gfCNCPoint3[2431] = {X 27.2875, Y 32.6686, Z -3.8333, A 0.000, B 0.000, C 0.000 }
gfCNCPoint3[2432] = {X 27.6591, Y 33.1493, Z -3.8333, A 0.000, B 0.000, C 0.000 }
gfCNCPoint3[2433] = {X 27.9609, Y 33.6765, Z -3.8333, A 0.000, B 0.000, C 0.000 }
gfCNCPoint3[2434] = {X 30.9820, Y 39.9182, Z -3.8333, A 0.000, B 0.000, C 0.000 }
gfCNCPoint3[2435] = {X 31.3085, Y 40.8441, Z -3.8333, A 0.000, B 0.000, C 0.000 }
gfCNCPoint3[2436] = {X 31.4215, Y 41.8194, Z -3.8333, A 0.000, B 0.000, C 0.000 }
gfCNCPoint3[2437] = {X 31.3155, Y 42.7955, Z -3.8333, A 0.000, B 0.000, C 0.000 }
gfCNCPoint3[2438] = {X 30.9956, Y 43.7238, Z -3.8333, A 0.000, B 0.000, C 0.000 }
gfCNCPoint3[2439] = {X 30.4779, Y 44.5580, Z -3.8333, A 0.000, B 0.000, C 0.000 }
gfCNCPoint3[2440] = {X 29.7880, Y 45.2567, Z -3.8333, A 0.000, B 0.000, C 0.000 }
gfCNCPoint3[2441] = {X 29.2517, Y 45.6903, Z -3.8333, A 0.000, B 0.000, C 0.000 }
gfCNCPoint3[2442] = {X 28.5404, Y 46.1589, Z -3.8333, A 0.000, B 0.000, C 0.000 }
gfCNCPoint3[2443] = {X 27.7524, Y 46.4822, Z -3.8333, A 0.000, B 0.000, C 0.000 }
gfCNCPoint3[2444] = {X 26.9169, Y 46.6482, Z -3.8333, A 0.000, B 0.000, C 0.000 }
gfCNCPoint3[2445] = {X 26.0652, Y 46.6506, Z -3.8333, A 0.000, B 0.000, C 0.000 }
gfCNCPoint3[2446] = {X 25.2288, Y 46.4895, Z -3.8333, A 0.000, B 0.000, C 0.000 }
gfCNCPoint3[2447] = {X 23.4341, Y 47.4359, Z -3.8333, A 0.000, B 0.000, C 0.000 }
gfCNCPoint3[2448] = {X 21.5778, Y 48.2550, Z -3.8333, A 0.000, B 0.000, C 0.000 }
gfCNCPoint3[2449] = {X 19.6689, Y 48.9428, Z -3.8333, A 0.000, B 0.000, C 0.000 }
gfCNCPoint3[2450] = {X 19.5102, Y 48.9962, Z -3.8333, A 0.000, B 0.000, C 0.000 }
gfCNCPoint3[2451] = {X 17.3375, Y 49.5790, Z -3.8333, A 0.000, B 0.000, C 0.000 }
gfCNCPoint3[2452] = {X 15.1180, Y 49.9462, Z -3.8333, A 0.000, B 0.000, C 0.000 }
gfCNCPoint3[2453] = {X 12.8733, Y 50.0942, Z -3.8333, A 0.000, B 0.000, C 0.000 }
gfCNCPoint3[2454] = {X 10.6249, Y 50.0215, Z -3.8333, A 0.000, B 0.000, C 0.000 }
gfCNCPoint3[2455] = {X 8.3945, Y 49.7289, Z -3.8333, A 0.000, B 0.000, C 0.000 }
gfCNCPoint3[2456] = {X 6.6781, Y 49.3407, Z -3.8333, A 0.000, B 0.000, C 0.000 }
gfCNCPoint3[2457] = {X 5.0104, Y 48.7788, Z -3.8333, A 0.000, B 0.000, C 0.000 }
gfCNCPoint3[2458] = {X 3.4090, Y 48.0493, Z -3.8333, A 0.000, B 0.000, C 0.000 }
gfCNCPoint3[2459] = {X 2.3280, Y 47.4375, Z -3.8333, A 0.000, B 0.000, C 0.000 }
gfCNCPoint3[2460] = {X 1.2941, Y 46.7491, Z -3.8333, A 0.000, B 0.000, C 0.000 }
gfCNCPoint3[2461] = {X 0.5975, Y 46.2081, Z -3.8333, A 0.000, B 0.000, C 0.000 }
gfCNCPoint3[2462] = {X -0.5424, Y 45.1839, Z -3.8333, A 0.000, B 0.000, C 0.000 }
gfCNCPoint3[2463] = {X -1.5547, Y 44.0333, Z -3.8333, A 0.000, B 0.000, C 0.000 }
gfCNCPoint3[2464] = {X -2.4254, Y 42.7723, Z -3.8333, A 0.000, B 0.000, C 0.000 }
gfCNCPoint3[2465] = {X -3.1426, Y 41.4180, Z -3.8333, A 0.000, B 0.000, C 0.000 }
gfCNCPoint3[2466] = {X -3.6965, Y 39.9892, Z -3.8333, A 0.000, B 0.000, C 0.000 }
gfCNCPoint3[2467] = {X -3.6965, Y 41.3532, Z -3.8333, A 0.000, B 0.000, C 0.000 }
gfCNCPoint3[2468] = {X -3.0110, Y 42.7243, Z -3.8333, A 0.000, B 0.000, C 0.000 }
gfCNCPoint3[2469] = {X -2.1750, Y 44.0092, Z -3.8333, A 0.000, B 0.000, C 0.000 }
gfCNCPoint3[2470] = {X -1.1994, Y 45.1915, Z -3.8333, A 0.000, B 0.000, C 0.000 }
gfCNCPoint3[2471] = {X -0.0965, Y 46.2561, Z -3.8333, A 0.000, B 0.000, C 0.000 }
gfCNCPoint3[2472] = {X -0.0965, Y 99.1431, Z -3.8333, A 0.000, B 0.000, C 0.000 }
gfCNCPoint3[2473] = {X -0.0948, Y 100.0187, Z -3.8333, A 0.000, B 0.000, C 0.000 }
gfCNCPoint3[2474] = {X -0.0672, Y 100.0698, Z -3.8333, A 0.000, B 0.000, C 0.000 }
gfCNCPoint3[2475] = {X -0.0148, Y 100.0950, Z -3.8333, A 0.000, B 0.000, C 0.000 }
gfCNCPoint3[2476] = {X 120.5926, Y 100.0950, Z -3.8333, A 0.000, B 0.000, C 0.000 }
gfCNCPoint3[2477] = {X 121.0613, Y 100.8812, Z -3.8333, A 0.000, B 0.000, C 0.000 }
gfCNCPoint3[2478] = {X 121.6687, Y 101.5660, Z -3.8333, A 0.000, B 0.000, C 0.000 }
gfCNCPoint3[2479] = {X 122.3932, Y 102.1254, Z -3.8333, A 0.000, B 0.000, C 0.000 }
gfCNCPoint3[2480] = {X 123.2094, Y 102.5396, Z -3.8333, A 0.000, B 0.000, C 0.000 }
gfCNCPoint3[2481] = {X 124.0887, Y 102.7942, Z -3.8333, A 0.000, B 0.000, C 0.000 }
gfCNCPoint3[2482] = {X 125.0000, Y 102.8800, Z -3.8333, A 0.000, B 0.000, C 0.000 }
gfCNCPoint3[2483] = {X 143.7791, Y 102.8800, Z -3.8333, A 0.000, B 0.000, C 0.000 }
gfCNCPoint3[2484] = {X 144.6904, Y 102.7942, Z -3.8333, A 0.000, B 0.000, C 0.000 }
gfCNCPoint3[2485] = {X 145.5697, Y 102.5396, Z -3.8333, A 0.000, B 0.000, C 0.000 }
gfCNCPoint3[2486] = {X 146.3859, Y 102.1254, Z -3.8333, A 0.000, B 0.000, C 0.000 }
gfCNCPoint3[2487] = {X 147.1104, Y 101.5660, Z -3.8333, A 0.000, B 0.000, C 0.000 }
gfCNCPoint3[2488] = {X 147.7178, Y 100.8812, Z -3.8333, A 0.000, B 0.000, C 0.000 }
gfCNCPoint3[2489] = {X 148.1865, Y 100.0950, Z -3.8333, A 0.000, B 0.000, C 0.000 }
gfCNCPoint3[2490] = {X 150.8375, Y 100.0950, Z -3.8333, A 0.000, B 0.000, C 0.000 }
gfCNCPoint3[2491] = {X 150.8375, Y 95.2950, Z -3.8333, A 0.000, B 0.000, C 0.000 }
gfCNCPoint3[2492] = {X 187.9256, Y 95.2950, Z -3.8333, A 0.000, B 0.000, C 0.000 }
gfCNCPoint3[2493] = {X 187.9777, Y 95.0990, Z -3.8333, A 0.000, B 0.000, C 0.000 }
gfCNCPoint3[2494] = {X 188.0352, Y 94.9045, Z -3.8333, A 0.000, B 0.000, C 0.000 }
gfCNCPoint3[2495] = {X 187.2619, Y 94.0602, Z -3.8333, A 0.000, B 0.000, C 0.000 }
gfCNCPoint3[2496] = {X 151.4055, Y 94.0602, Z -3.8333, A 0.000, B 0.000, C 0.000 }
gfCNCPoint3[2497] = {X 150.7056, Y 94.8356, Z -3.8333, A 0.000, B 0.000, C 0.000 }
gfCNCPoint3[2498] = {X 150.7753, Y 95.0642, Z -3.8333, A 0.000, B 0.000, C 0.000 }
gfCNCPoint3[2499] = {X 150.8375, Y 95.2950, Z -3.8333, A 0.000, B 0.000, C 0.000 }
gfCNCPoint3[2500] = {X 150.8375, Y 97.6950, Z -3.8333, A 0.000, B 0.000, C 0.000 }
gfCNCPoint3[2501] = {X 190.1070, Y 97.6950, Z -3.8333, A 0.000, B 0.000, C 0.000 }
gfCNCPoint3[2502] = {X 190.1070, Y 97.0659, Z -3.8333, A 0.000, B 0.000, C 0.000 }
gfCNCPoint3[2503] = {X 190.1938, Y 96.1495, Z -3.8333, A 0.000, B 0.000, C 0.000 }
gfCNCPoint3[2504] = {X 190.4511, Y 95.2657, Z -3.8333, A 0.000, B 0.000, C 0.000 }
gfCNCPoint3[2505] = {X 190.8699, Y 94.4460, Z -3.8333, A 0.000, B 0.000, C 0.000 }
gfCNCPoint3[2506] = {X 188.3182, Y 91.6602, Z -3.8333, A 0.000, B 0.000, C 0.000 }
gfCNCPoint3[2507] = {X 150.3387, Y 91.6602, Z -3.8333, A 0.000, B 0.000, C 0.000 }
gfCNCPoint3[2508] = {X 147.8637, Y 94.4023, Z -3.8333, A 0.000, B 0.000, C 0.000 }
gfCNCPoint3[2509] = {X 148.2978, Y 95.2327, Z -3.8333, A 0.000, B 0.000, C 0.000 }
gfCNCPoint3[2510] = {X 148.5662, Y 96.1304, Z -3.8333, A 0.000, B 0.000, C 0.000 }
gfCNCPoint3[2511] = {X 148.6591, Y 97.0628, Z -3.8333, A 0.000, B 0.000, C 0.000 }
gfCNCPoint3[2512] = {X 148.6591, Y 97.6950, Z -3.8333, A 0.000, B 0.000, C 0.000 }
gfCNCPoint3[2513] = {X 150.8375, Y 97.6950, Z -3.8333, A 0.000, B 0.000, C 0.000 }
gfCNCPoint3[2514] = {X 150.8375, Y 100.0950, Z -3.8333, A 0.000, B 0.000, C 0.000 }
gfCNCPoint3[2515] = {X 190.5795, Y 100.0950, Z -3.8333, A 0.000, B 0.000, C 0.000 }
gfCNCPoint3[2516] = {X 191.0483, Y 100.8812, Z -3.8333, A 0.000, B 0.000, C 0.000 }
gfCNCPoint3[2517] = {X 191.6556, Y 101.5660, Z -3.8333, A 0.000, B 0.000, C 0.000 }
gfCNCPoint3[2518] = {X 192.3802, Y 102.1254, Z -3.8333, A 0.000, B 0.000, C 0.000 }
gfCNCPoint3[2519] = {X 193.1964, Y 102.5396, Z -3.8333, A 0.000, B 0.000, C 0.000 }
gfCNCPoint3[2520] = {X 194.0757, Y 102.7942, Z -3.8333, A 0.000, B 0.000, C 0.000 }
gfCNCPoint3[2521] = {X 194.9870, Y 102.8800, Z -3.8333, A 0.000, B 0.000, C 0.000 }
gfCNCPoint3[2522] = {X 212.6141, Y 102.8800, Z -3.8333, A 0.000, B 0.000, C 0.000 }
gfCNCPoint3[2523] = {X 213.0066, Y 102.8642, Z -3.8333, A 0.000, B 0.000, C 0.000 }
gfCNCPoint3[2524] = {X 213.3966, Y 102.8169, Z -3.8333, A 0.000, B 0.000, C 0.000 }
gfCNCPoint3[2525] = {X 213.7865, Y 102.8642, Z -3.8333, A 0.000, B 0.000, C 0.000 }
gfCNCPoint3[2526] = {X 214.1790, Y 102.8800, Z -3.8333, A 0.000, B 0.000, C 0.000 }
gfCNCPoint3[2527] = {X 233.4798, Y 102.8800, Z -3.8333, A 0.000, B 0.000, C 0.000 }
gfCNCPoint3[2528] = {X 234.3911, Y 102.7942, Z -3.8333, A 0.000, B 0.000, C 0.000 }
gfCNCPoint3[2529] = {X 235.2703, Y 102.5396, Z -3.8333, A 0.000, B 0.000, C 0.000 }
gfCNCPoint3[2530] = {X 236.0866, Y 102.1254, Z -3.8333, A 0.000, B 0.000, C 0.000 }
gfCNCPoint3[2531] = {X 236.8111, Y 101.5660, Z -3.8333, A 0.000, B 0.000, C 0.000 }
gfCNCPoint3[2532] = {X 237.4185, Y 100.8812, Z -3.8333, A 0.000, B 0.000, C 0.000 }
gfCNCPoint3[2533] = {X 237.8872, Y 100.0950, Z -3.8333, A 0.000, B 0.000, C 0.000 }
gfCNCPoint3[2534] = {X 261.4774, Y 100.0950, Z -3.8333, A 0.000, B 0.000, C 0.000 }
gfCNCPoint3[2535] = {X 261.4774, Y 90.4950, Z -3.8333, A 0.000, B 0.000, C 0.000 }
gfCNCPoint3[2536] = {X 266.0962, Y 90.4950, Z -3.8333, A 0.000, B 0.000, C 0.000 }
gfCNCPoint3[2537] = {X 266.1752, Y 90.3747, Z -3.8333, A 0.000, B 0.000, C 0.000 }
gfCNCPoint3[2538] = {X 266.2556, Y 90.2554, Z -3.8333, A 0.000, B 0.000, C 0.000 }
gfCNCPoint3[2539] = {X 263.5094, Y 89.1788, Z -3.8333, A 0.000, B 0.000, C 0.000 }
gfCNCPoint3[2540] = {X 261.4774, Y 90.4950, Z -3.8333, A 0.000, B 0.000, C 0.000 }
gfCNCPoint3[2541] = {X 261.4774, Y 92.8950, Z -3.8333, A 0.000, B 0.000, C 0.000 }
gfCNCPoint3[2542] = {X 267.4974, Y 92.8950, Z -3.8333, A 0.000, B 0.000, C 0.000 }
gfCNCPoint3[2543] = {X 267.8429, Y 92.2375, Z -3.8333, A 0.000, B 0.000, C 0.000 }
gfCNCPoint3[2544] = {X 268.2378, Y 91.6085, Z -3.8333, A 0.000, B 0.000, C 0.000 }
gfCNCPoint3[2545] = {X 269.1700, Y 90.4463, Z -3.8333, A 0.000, B 0.000, C 0.000 }
gfCNCPoint3[2546] = {X 270.2694, Y 89.4409, Z -3.8333, A 0.000, B 0.000, C 0.000 }
gfCNCPoint3[2547] = {X 270.2694, Y 89.2510, Z -3.8333, A 0.000, B 0.000, C 0.000 }
gfCNCPoint3[2548] = {X 263.2385, Y 86.4948, Z -3.8333, A 0.000, B 0.000, C 0.000 }
gfCNCPoint3[2549] = {X 253.3574, Y 92.8950, Z -3.8333, A 0.000, B 0.000, C 0.000 }
gfCNCPoint3[2550] = {X 261.4774, Y 92.8950, Z -3.8333, A 0.000, B 0.000, C 0.000 }
gfCNCPoint3[2551] = {X 261.4774, Y 95.2950, Z -3.8333, A 0.000, B 0.000, C 0.000 }
gfCNCPoint3[2552] = {X 269.1714, Y 95.2950, Z -3.8333, A 0.000, B 0.000, C 0.000 }
gfCNCPoint3[2553] = {X 269.5516, Y 94.1744, Z -3.8333, A 0.000, B 0.000, C 0.000 }
gfCNCPoint3[2554] = {X 270.1082, Y 93.1303, Z -3.8333, A 0.000, B 0.000, C 0.000 }
gfCNCPoint3[2555] = {X 270.8267, Y 92.1901, Z -3.8333, A 0.000, B 0.000, C 0.000 }
gfCNCPoint3[2556] = {X 271.6880, Y 91.3787, Z -3.8333, A 0.000, B 0.000, C 0.000 }
gfCNCPoint3[2557] = {X 272.6694, Y 90.7176, Z -3.8333, A 0.000, B 0.000, C 0.000 }
gfCNCPoint3[2558] = {X 272.6694, Y 87.6139, Z -3.8333, A 0.000, B 0.000, C 0.000 }
gfCNCPoint3[2559] = {X 262.9676, Y 83.8108, Z -3.8333, A 0.000, B 0.000, C 0.000 }
gfCNCPoint3[2560] = {X 245.2375, Y 95.2950, Z -3.8333, A 0.000, B 0.000, C 0.000 }
gfCNCPoint3[2561] = {X 261.4774, Y 95.2950, Z -3.8333, A 0.000, B 0.000, C 0.000 }
gfCNCPoint3[2562] = {X 261.4774, Y 97.6950, Z -3.8333, A 0.000, B 0.000, C 0.000 }
gfCNCPoint3[2563] = {X 271.3527, Y 97.6950, Z -3.8333, A 0.000, B 0.000, C 0.000 }
gfCNCPoint3[2564] = {X 271.3529, Y 97.0186, Z -3.8333, A 0.000, B 0.000, C 0.000 }
gfCNCPoint3[2565] = {X 271.4810, Y 95.9545, Z -3.8333, A 0.000, B 0.000, C 0.000 }
gfCNCPoint3[2566] = {X 271.8382, Y 94.9440, Z -3.8333, A 0.000, B 0.000, C 0.000 }
gfCNCPoint3[2567] = {X 272.4073, Y 94.0359, Z -3.8333, A 0.000, B 0.000, C 0.000 }
gfCNCPoint3[2568] = {X 273.1610, Y 93.2739, Z -3.8333, A 0.000, B 0.000, C 0.000 }
gfCNCPoint3[2569] = {X 274.0629, Y 92.6949, Z -3.8333, A 0.000, B 0.000, C 0.000 }
gfCNCPoint3[2570] = {X 275.0694, Y 92.3266, Z -3.8333, A 0.000, B 0.000, C 0.000 }
gfCNCPoint3[2571] = {X 275.0694, Y 85.9769, Z -3.8333, A 0.000, B 0.000, C 0.000 }
gfCNCPoint3[2572] = {X 262.6987, Y 81.1276, Z -3.8333, A 0.000, B 0.000, C 0.000 }
gfCNCPoint3[2573] = {X 262.5781, Y 81.2036, Z -3.8333, A 0.000, B 0.000, C 0.000 }
gfCNCPoint3[2574] = {X 238.3586, Y 96.8912, Z -3.8333, A 0.000, B 0.000, C 0.000 }
gfCNCPoint3[2575] = {X 238.3598, Y 97.0659, Z -3.8333, A 0.000, B 0.000, C 0.000 }
gfCNCPoint3[2576] = {X 238.3598, Y 97.6950, Z -3.8333, A 0.000, B 0.000, C 0.000 }
gfCNCPoint3[2577] = {X 261.4774, Y 97.6950, Z -3.8333, A 0.000, B 0.000, C 0.000 }
gfCNCPoint3[2578] = {X 261.4774, Y 100.0950, Z -3.8333, A 0.000, B 0.000, C 0.000 }
gfCNCPoint3[2579] = {X 271.8253, Y 100.0950, Z -3.8333, A 0.000, B 0.000, C 0.000 }
gfCNCPoint3[2580] = {X 272.2940, Y 100.8812, Z -3.8333, A 0.000, B 0.000, C 0.000 }
gfCNCPoint3[2581] = {X 272.9014, Y 101.5660, Z -3.8333, A 0.000, B 0.000, C 0.000 }
gfCNCPoint3[2582] = {X 273.6259, Y 102.1254, Z -3.8333, A 0.000, B 0.000, C 0.000 }
gfCNCPoint3[2583] = {X 274.4421, Y 102.5396, Z -3.8333, A 0.000, B 0.000, C 0.000 }
gfCNCPoint3[2584] = {X 275.3214, Y 102.7942, Z -3.8333, A 0.000, B 0.000, C 0.000 }
gfCNCPoint3[2585] = {X 276.2327, Y 102.8800, Z -3.8333, A 0.000, B 0.000, C 0.000 }
gfCNCPoint3[2586] = {X 292.7731, Y 102.8800, Z -3.8333, A 0.000, B 0.000, C 0.000 }
gfCNCPoint3[2587] = {X 293.6844, Y 102.7942, Z -3.8333, A 0.000, B 0.000, C 0.000 }
gfCNCPoint3[2588] = {X 294.5636, Y 102.5396, Z -3.8333, A 0.000, B 0.000, C 0.000 }
gfCNCPoint3[2589] = {X 295.3799, Y 102.1254, Z -3.8333, A 0.000, B 0.000, C 0.000 }
gfCNCPoint3[2590] = {X 296.1044, Y 101.5660, Z -3.8333, A 0.000, B 0.000, C 0.000 }
gfCNCPoint3[2591] = {X 296.7118, Y 100.8812, Z -3.8333, A 0.000, B 0.000, C 0.000 }
gfCNCPoint3[2592] = {X 297.1805, Y 100.0950, Z -3.8333, A 0.000, B 0.000, C 0.000 }
gfCNCPoint3[2593] = {X 319.1331, Y 100.0950, Z -3.8333, A 0.000, B 0.000, C 0.000 }
gfCNCPoint3[2594] = {X 321.4361, Y 100.8684, Z -3.8333, A 0.000, B 0.000, C 0.000 }
gfCNCPoint3[2595] = {X 323.7818, Y 101.5002, Z -3.8333, A 0.000, B 0.000, C 0.000 }
gfCNCPoint3[2596] = {X 326.1617, Y 101.9882, Z -3.8333, A 0.000, B 0.000, C 0.000 }
gfCNCPoint3[2597] = {X 329.6399, Y 102.5404, Z -3.8333, A 0.000, B 0.000, C 0.000 }
gfCNCPoint3[2598] = {X 333.1372, Y 102.9558, Z -3.8333, A 0.000, B 0.000, C 0.000 }
gfCNCPoint3[2599] = {X 336.6480, Y 103.2337, Z -3.8333, A 0.000, B 0.000, C 0.000 }
gfCNCPoint3[2600] = {X 342.8090, Y 103.5157, Z -3.8333, A 0.000, B 0.000, C 0.000 }
gfCNCPoint3[2601] = {X 348.9760, Y 103.5923, Z -3.8333, A 0.000, B 0.000, C 0.000 }
gfCNCPoint3[2602] = {X 355.1421, Y 103.4635, Z -3.8333, A 0.000, B 0.000, C 0.000 }
gfCNCPoint3[2603] = {X 361.3005, Y 103.1293, Z -3.8333, A 0.000, B 0.000, C 0.000 }
gfCNCPoint3[2604] = {X 365.1928, Y 102.7587, Z -3.8333, A 0.000, B 0.000, C 0.000 }
gfCNCPoint3[2605] = {X 369.0628, Y 102.2014, Z -3.8333, A 0.000, B 0.000, C 0.000 }
gfCNCPoint3[2606] = {X 372.9015, Y 101.4586, Z -3.8333, A 0.000, B 0.000, C 0.000 }
gfCNCPoint3[2607] = {X 375.2301, Y 100.8565, Z -3.8333, A 0.000, B 0.000, C 0.000 }
gfCNCPoint3[2608] = {X 377.5115, Y 100.0950, Z -3.8333, A 0.000, B 0.000, C 0.000 }
gfCNCPoint3[2609] = {X 391.9985, Y 100.0950, Z -3.8333, A 0.000, B 0.000, C 0.000 }
gfCNCPoint3[2610] = {X 392.4673, Y 100.8812, Z -3.8333, A 0.000, B 0.000, C 0.000 }
gfCNCPoint3[2611] = {X 393.0746, Y 101.5660, Z -3.8333, A 0.000, B 0.000, C 0.000 }
gfCNCPoint3[2612] = {X 393.7991, Y 102.1254, Z -3.8333, A 0.000, B 0.000, C 0.000 }
gfCNCPoint3[2613] = {X 394.6154, Y 102.5396, Z -3.8333, A 0.000, B 0.000, C 0.000 }
gfCNCPoint3[2614] = {X 395.4946, Y 102.7942, Z -3.8333, A 0.000, B 0.000, C 0.000 }
gfCNCPoint3[2615] = {X 396.4059, Y 102.8800, Z -3.8333, A 0.000, B 0.000, C 0.000 }
gfCNCPoint3[2616] = {X 415.7067, Y 102.8800, Z -3.8333, A 0.000, B 0.000, C 0.000 }
gfCNCPoint3[2617] = {X 416.6180, Y 102.7942, Z -3.8333, A 0.000, B 0.000, C 0.000 }
gfCNCPoint3[2618] = {X 417.4973, Y 102.5396, Z -3.8333, A 0.000, B 0.000, C 0.000 }
gfCNCPoint3[2619] = {X 418.3135, Y 102.1254, Z -3.8333, A 0.000, B 0.000, C 0.000 }
gfCNCPoint3[2620] = {X 419.0380, Y 101.5660, Z -3.8333, A 0.000, B 0.000, C 0.000 }
gfCNCPoint3[2621] = {X 419.6454, Y 100.8812, Z -3.8333, A 0.000, B 0.000, C 0.000 }
gfCNCPoint3[2622] = {X 420.1141, Y 100.0950, Z -3.8333, A 0.000, B 0.000, C 0.000 }
gfCNCPoint3[2623] = {X 443.7023, Y 100.0950, Z -3.8333, A 0.000, B 0.000, C 0.000 }
gfCNCPoint3[2624] = {X 443.7023, Y 90.4950, Z -3.8333, A 0.000, B 0.000, C 0.000 }
gfCNCPoint3[2625] = {X 448.3231, Y 90.4950, Z -3.8333, A 0.000, B 0.000, C 0.000 }
gfCNCPoint3[2626] = {X 448.4021, Y 90.3747, Z -3.8333, A 0.000, B 0.000, C 0.000 }
gfCNCPoint3[2627] = {X 448.4825, Y 90.2554, Z -3.8333, A 0.000, B 0.000, C 0.000 }
gfCNCPoint3[2628] = {X 445.7349, Y 89.1783, Z -3.8333, A 0.000, B 0.000, C 0.000 }
gfCNCPoint3[2629] = {X 443.7023, Y 90.4950, Z -3.8333, A 0.000, B 0.000, C 0.000 }
gfCNCPoint3[2630] = {X 443.7023, Y 92.8950, Z -3.8333, A 0.000, B 0.000, C 0.000 }
gfCNCPoint3[2631] = {X 449.7243, Y 92.8950, Z -3.8333, A 0.000, B 0.000, C 0.000 }
gfCNCPoint3[2632] = {X 450.0698, Y 92.2375, Z -3.8333, A 0.000, B 0.000, C 0.000 }
gfCNCPoint3[2633] = {X 450.4647, Y 91.6084, Z -3.8333, A 0.000, B 0.000, C 0.000 }
gfCNCPoint3[2634] = {X 451.3969, Y 90.4463, Z -3.8333, A 0.000, B 0.000, C 0.000 }
gfCNCPoint3[2635] = {X 452.4963, Y 89.4409, Z -3.8333, A 0.000, B 0.000, C 0.000 }
gfCNCPoint3[2636] = {X 452.4963, Y 89.2510, Z -3.8333, A 0.000, B 0.000, C 0.000 }
gfCNCPoint3[2637] = {X 445.4640, Y 86.4943, Z -3.8333, A 0.000, B 0.000, C 0.000 }
gfCNCPoint3[2638] = {X 435.5831, Y 92.8950, Z -3.8333, A 0.000, B 0.000, C 0.000 }
gfCNCPoint3[2639] = {X 443.7023, Y 92.8950, Z -3.8333, A 0.000, B 0.000, C 0.000 }
gfCNCPoint3[2640] = {X 443.7023, Y 95.2950, Z -3.8333, A 0.000, B 0.000, C 0.000 }
gfCNCPoint3[2641] = {X 451.3983, Y 95.2950, Z -3.8333, A 0.000, B 0.000, C 0.000 }
gfCNCPoint3[2642] = {X 451.7785, Y 94.1744, Z -3.8333, A 0.000, B 0.000, C 0.000 }
gfCNCPoint3[2643] = {X 452.3351, Y 93.1303, Z -3.8333, A 0.000, B 0.000, C 0.000 }
gfCNCPoint3[2644] = {X 453.0536, Y 92.1901, Z -3.8333, A 0.000, B 0.000, C 0.000 }
gfCNCPoint3[2645] = {X 453.9149, Y 91.3787, Z -3.8333, A 0.000, B 0.000, C 0.000 }
gfCNCPoint3[2646] = {X 454.8963, Y 90.7176, Z -3.8333, A 0.000, B 0.000, C 0.000 }
gfCNCPoint3[2647] = {X 454.8963, Y 87.6139, Z -3.8333, A 0.000, B 0.000, C 0.000 }
gfCNCPoint3[2648] = {X 445.1930, Y 83.8102, Z -3.8333, A 0.000, B 0.000, C 0.000 }
gfCNCPoint3[2649] = {X 427.4639, Y 95.2950, Z -3.8333, A 0.000, B 0.000, C 0.000 }
gfCNCPoint3[2650] = {X 443.7023, Y 95.2950, Z -3.8333, A 0.000, B 0.000, C 0.000 }
gfCNCPoint3[2651] = {X 443.7023, Y 97.6950, Z -3.8333, A 0.000, B 0.000, C 0.000 }
gfCNCPoint3[2652] = {X 453.5796, Y 97.6950, Z -3.8333, A 0.000, B 0.000, C 0.000 }
gfCNCPoint3[2653] = {X 453.5796, Y 97.0659, Z -3.8333, A 0.000, B 0.000, C 0.000 }
gfCNCPoint3[2654] = {X 453.6990, Y 95.9930, Z -3.8333, A 0.000, B 0.000, C 0.000 }
gfCNCPoint3[2655] = {X 454.0514, Y 94.9725, Z -3.8333, A 0.000, B 0.000, C 0.000 }
gfCNCPoint3[2656] = {X 454.6196, Y 94.0545, Z -3.8333, A 0.000, B 0.000, C 0.000 }
gfCNCPoint3[2657] = {X 455.3757, Y 93.2839, Z -3.8333, A 0.000, B 0.000, C 0.000 }
gfCNCPoint3[2658] = {X 456.2827, Y 92.6984, Z -3.8333, A 0.000, B 0.000, C 0.000 }
gfCNCPoint3[2659] = {X 457.2963, Y 92.3266, Z -3.8333, A 0.000, B 0.000, C 0.000 }
gfCNCPoint3[2660] = {X 457.2963, Y 85.9769, Z -3.8333, A 0.000, B 0.000, C 0.000 }
gfCNCPoint3[2661] = {X 444.9220, Y 81.1262, Z -3.8333, A 0.000, B 0.000, C 0.000 }
gfCNCPoint3[2662] = {X 420.5854, Y 96.8912, Z -3.8333, A 0.000, B 0.000, C 0.000 }
gfCNCPoint3[2663] = {X 420.5867, Y 97.0659, Z -3.8333, A 0.000, B 0.000, C 0.000 }
gfCNCPoint3[2664] = {X 420.5867, Y 97.6950, Z -3.8333, A 0.000, B 0.000, C 0.000 }
gfCNCPoint3[2665] = {X 443.7023, Y 97.6950, Z -3.8333, A 0.000, B 0.000, C 0.000 }
gfCNCPoint3[2666] = {X 443.7023, Y 100.0950, Z -3.8333, A 0.000, B 0.000, C 0.000 }
gfCNCPoint3[2667] = {X 454.0522, Y 100.0950, Z -3.8333, A 0.000, B 0.000, C 0.000 }
gfCNCPoint3[2668] = {X 454.5209, Y 100.8812, Z -3.8333, A 0.000, B 0.000, C 0.000 }
gfCNCPoint3[2669] = {X 455.1283, Y 101.5660, Z -3.8333, A 0.000, B 0.000, C 0.000 }
gfCNCPoint3[2670] = {X 455.8528, Y 102.1254, Z -3.8333, A 0.000, B 0.000, C 0.000 }
gfCNCPoint3[2671] = {X 456.6691, Y 102.5396, Z -3.8333, A 0.000, B 0.000, C 0.000 }
gfCNCPoint3[2672] = {X 457.5483, Y 102.7942, Z -3.8333, A 0.000, B 0.000, C 0.000 }
gfCNCPoint3[2673] = {X 458.4596, Y 102.8800, Z -3.8333, A 0.000, B 0.000, C 0.000 }
gfCNCPoint3[2674] = {X 475.0000, Y 102.8800, Z -3.8333, A 0.000, B 0.000, C 0.000 }
gfCNCPoint3[2675] = {X 475.9113, Y 102.7942, Z -3.8333, A 0.000, B 0.000, C 0.000 }
gfCNCPoint3[2676] = {X 476.7906, Y 102.5396, Z -3.8333, A 0.000, B 0.000, C 0.000 }
gfCNCPoint3[2677] = {X 477.6068, Y 102.1254, Z -3.8333, A 0.000, B 0.000, C 0.000 }
gfCNCPoint3[2678] = {X 478.3313, Y 101.5660, Z -3.8333, A 0.000, B 0.000, C 0.000 }
gfCNCPoint3[2679] = {X 478.9387, Y 100.8812, Z -3.8333, A 0.000, B 0.000, C 0.000 }
gfCNCPoint3[2680] = {X 479.4074, Y 100.0950, Z -3.8333, A 0.000, B 0.000, C 0.000 }
gfCNCPoint3[2681] = {X 507.6816, Y 100.0950, Z -3.8333, A 0.000, B 0.000, C 0.000 }
gfCNCPoint3[2682] = {X 507.6816, Y 107.6950, Z -3.8333, A 0.000, B 0.000, C 0.000 }
gfCNCPoint3[2683] = {X 507.6816, Y 107.6950, Z -0.8333, A 0.000, B 0.000, C 0.000 }
gfCNCPoint3[2684] = {X 507.6816, Y 107.6950, Z 11.0000, A 0.000, B 0.000, C 0.000 }
gfCNCPoint3[2685] = {X 108.5561, Y 40.8996, Z 11.0000, A 0.000, B 0.000, C 0.000 }
gfCNCPoint3[2686] = {X 108.5561, Y 40.8996, Z 0.0000, A 0.000, B 0.000, C 0.000 }
gfCNCPoint3[2687] = {X 108.5561, Y 40.8996, Z -3.8333, A 0.000, B 0.000, C 0.000 }
gfCNCPoint3[2688] = {X 108.0660, Y 42.0973, Z -3.8333, A 0.000, B 0.000, C 0.000 }
gfCNCPoint3[2689] = {X 108.0932, Y 42.0499, Z -3.8333, A 0.000, B 0.000, C 0.000 }
gfCNCPoint3[2690] = {X 108.1209, Y 42.0029, Z -3.8333, A 0.000, B 0.000, C 0.000 }
gfCNCPoint3[2691] = {X 108.5462, Y 41.3863, Z -3.8333, A 0.000, B 0.000, C 0.000 }
gfCNCPoint3[2692] = {X 109.0463, Y 40.8285, Z -3.8333, A 0.000, B 0.000, C 0.000 }
gfCNCPoint3[2693] = {X 109.0462, Y 39.7020, Z -3.8333, A 0.000, B 0.000, C 0.000 }
gfCNCPoint3[2694] = {X 108.5561, Y 40.8996, Z -3.8333, A 0.000, B 0.000, C 0.000 }
gfCNCPoint3[2695] = {X 108.5561, Y 40.8996, Z -0.8333, A 0.000, B 0.000, C 0.000 }
gfCNCPoint3[2696] = {X 108.5561, Y 40.8996, Z 11.0000, A 0.000, B 0.000, C 0.000 }
gfCNCPoint3[2697] = {X 95.6836, Y 40.8744, Z 11.0000, A 0.000, B 0.000, C 0.000 }
gfCNCPoint3[2698] = {X 95.6836, Y 40.8744, Z 0.0000, A 0.000, B 0.000, C 0.000 }
gfCNCPoint3[2699] = {X 95.6836, Y 40.8744, Z -3.8333, A 0.000, B 0.000, C 0.000 }
gfCNCPoint3[2700] = {X 95.2107, Y 39.7180, Z -3.8333, A 0.000, B 0.000, C 0.000 }
gfCNCPoint3[2701] = {X 95.2108, Y 40.8688, Z -3.8333, A 0.000, B 0.000, C 0.000 }
gfCNCPoint3[2702] = {X 95.7325, Y 41.4100, Z -3.8333, A 0.000, B 0.000, C 0.000 }
gfCNCPoint3[2703] = {X 96.1564, Y 42.0308, Z -3.8333, A 0.000, B 0.000, C 0.000 }
gfCNCPoint3[2704] = {X 95.6836, Y 40.8744, Z -3.8333, A 0.000, B 0.000, C 0.000 }
gfCNCPoint3[2705] = {X 95.6836, Y 40.8744, Z -0.8333, A 0.000, B 0.000, C 0.000 }
gfCNCPoint3[2706] = {X 95.6836, Y 40.8744, Z 11.0000, A 0.000, B 0.000, C 0.000 }
gfCNCPoint3[2707] = {X -7.6965, Y 43.3001, Z 11.0000, A 0.000, B 0.000, C 0.000 }
gfCNCPoint3[2708] = {X -7.6965, Y 43.3001, Z -0.8333, A 0.000, B 0.000, C 0.000 }
gfCNCPoint3[2709] = {X -7.6965, Y 43.3001, Z -3.8333, A 0.000, B 0.000, C 0.000 }
gfCNCPoint3[2710] = {X -3.6965, Y 30.8026, Z -3.8333, A 0.000, B 0.000, C 0.000 }
gfCNCPoint3[2711] = {X -3.5205, Y 30.2854, Z -3.8333, A 0.000, B 0.000, C 0.000 }
gfCNCPoint3[2712] = {X -3.3256, Y 29.7750, Z -3.8333, A 0.000, B 0.000, C 0.000 }
gfCNCPoint3[2713] = {X -2.7025, Y 28.4549, Z -3.8333, A 0.000, B 0.000, C 0.000 }
gfCNCPoint3[2714] = {X -1.9088, Y 27.2299, Z -3.8333, A 0.000, B 0.000, C 0.000 }
gfCNCPoint3[2715] = {X -0.9586, Y 26.1219, Z -3.8333, A 0.000, B 0.000, C 0.000 }
gfCNCPoint3[2716] = {X 0.1311, Y 25.1507, Z -3.8333, A 0.000, B 0.000, C 0.000 }
gfCNCPoint3[2717] = {X 1.3407, Y 24.3338, Z -3.8333, A 0.000, B 0.000, C 0.000 }
gfCNCPoint3[2718] = {X 0.5801, Y 23.9235, Z -3.8333, A 0.000, B 0.000, C 0.000 }
gfCNCPoint3[2719] = {X -0.0857, Y 23.3725, Z -3.8333, A 0.000, B 0.000, C 0.000 }
gfCNCPoint3[2720] = {X -0.6309, Y 22.7020, Z -3.8333, A 0.000, B 0.000, C 0.000 }
gfCNCPoint3[2721] = {X -1.0345, Y 21.9378, Z -3.8333, A 0.000, B 0.000, C 0.000 }
gfCNCPoint3[2722] = {X -3.6458, Y 15.5423, Z -3.8333, A 0.000, B 0.000, C 0.000 }
gfCNCPoint3[2723] = {X -3.6717, Y 15.4774, Z -3.8333, A 0.000, B 0.000, C 0.000 }
gfCNCPoint3[2724] = {X -3.6965, Y 15.4121, Z -3.8333, A 0.000, B 0.000, C 0.000 }
gfCNCPoint3[2725] = {X -7.6965, Y 4.6502, Z -3.8333, A 0.000, B 0.000, C 0.000 }
gfCNCPoint3[2726] = {X -7.6965, Y 4.6502, Z -0.8333, A 0.000, B 0.000, C 0.000 }
gfCNCPoint3[2727] = {X -7.6965, Y 4.6502, Z 11.0000, A 0.000, B 0.000, C 0.000 }
gfCNCPoint3[2728] = {X -7.6965, Y 16.4125, Z 11.0000, A 0.000, B 0.000, C 0.000 }
gfCNCPoint3[2729] = {X -7.6965, Y 16.4125, Z -0.8333, A 0.000, B 0.000, C 0.000 }
gfCNCPoint3[2730] = {X -7.6965, Y 16.4125, Z -3.8333, A 0.000, B 0.000, C 0.000 }
gfCNCPoint3[2731] = {X -4.8868, Y 16.4125, Z -3.8333, A 0.000, B 0.000, C 0.000 }
gfCNCPoint3[2732] = {X -3.6965, Y 12.5937, Z -3.8333, A 0.000, B 0.000, C 0.000 }
gfCNCPoint3[2733] = {X -3.6605, Y 12.4834, Z -3.8333, A 0.000, B 0.000, C 0.000 }
gfCNCPoint3[2734] = {X -3.6216, Y 12.3740, Z -3.8333, A 0.000, B 0.000, C 0.000 }
gfCNCPoint3[2735] = {X -3.1666, Y 11.4828, Z -3.8333, A 0.000, B 0.000, C 0.000 }
gfCNCPoint3[2736] = {X -2.5188, Y 10.7200, Z -3.8333, A 0.000, B 0.000, C 0.000 }
gfCNCPoint3[2737] = {X -1.7129, Y 10.1268, Z -3.8333, A 0.000, B 0.000, C 0.000 }
gfCNCPoint3[2738] = {X -1.1157, Y 9.7861, Z -3.8333, A 0.000, B 0.000, C 0.000 }
gfCNCPoint3[2739] = {X -0.2296, Y 9.4046, Z -3.8333, A 0.000, B 0.000, C 0.000 }
gfCNCPoint3[2740] = {X 0.7191, Y 9.2293, Z -3.8333, A 0.000, B 0.000, C 0.000 }
gfCNCPoint3[2741] = {X 1.6830, Y 9.2689, Z -3.8333, A 0.000, B 0.000, C 0.000 }
gfCNCPoint3[2742] = {X 2.6141, Y 9.5214, Z -3.8333, A 0.000, B 0.000, C 0.000 }
gfCNCPoint3[2743] = {X 3.3937, Y 9.1539, Z -3.8333, A 0.000, B 0.000, C 0.000 }
gfCNCPoint3[2744] = {X 4.1978, Y 8.8435, Z -3.8333, A 0.000, B 0.000, C 0.000 }
gfCNCPoint3[2745] = {X 6.1085, Y 8.1749, Z -3.8333, A 0.000, B 0.000, C 0.000 }
gfCNCPoint3[2746] = {X 8.0697, Y 7.6735, Z -3.8333, A 0.000, B 0.000, C 0.000 }
gfCNCPoint3[2747] = {X 10.0669, Y 7.3431, Z -3.8333, A 0.000, B 0.000, C 0.000 }
gfCNCPoint3[2748] = {X 12.0851, Y 7.1861, Z -3.8333, A 0.000, B 0.000, C 0.000 }
gfCNCPoint3[2749] = {X 14.1093, Y 7.2037, Z -3.8333, A 0.000, B 0.000, C 0.000 }
gfCNCPoint3[2750] = {X 16.1245, Y 7.3958, Z -3.8333, A 0.000, B 0.000, C 0.000 }
gfCNCPoint3[2751] = {X 17.9477, Y 7.7294, Z -3.8333, A 0.000, B 0.000, C 0.000 }
gfCNCPoint3[2752] = {X 19.7252, Y 8.2544, Z -3.8333, A 0.000, B 0.000, C 0.000 }
gfCNCPoint3[2753] = {X 21.4370, Y 8.9650, Z -3.8333, A 0.000, B 0.000, C 0.000 }
gfCNCPoint3[2754] = {X 23.0638, Y 9.8531, Z -3.8333, A 0.000, B 0.000, C 0.000 }
gfCNCPoint3[2755] = {X 24.5873, Y 10.9087, Z -3.8333, A 0.000, B 0.000, C 0.000 }
gfCNCPoint3[2756] = {X 25.6726, Y 11.8575, Z -3.8333, A 0.000, B 0.000, C 0.000 }
gfCNCPoint3[2757] = {X 26.6461, Y 12.9206, Z -3.8333, A 0.000, B 0.000, C 0.000 }
gfCNCPoint3[2758] = {X 27.4958, Y 14.0851, Z -3.8333, A 0.000, B 0.000, C 0.000 }
gfCNCPoint3[2759] = {X 28.2113, Y 15.3364, Z -3.8333, A 0.000, B 0.000, C 0.000 }
gfCNCPoint3[2760] = {X 28.7839, Y 16.6594, Z -3.8333, A 0.000, B 0.000, C 0.000 }
gfCNCPoint3[2761] = {X 29.2584, Y 18.3158, Z -3.8333, A 0.000, B 0.000, C 0.000 }
gfCNCPoint3[2762] = {X 29.5400, Y 20.0156, Z -3.8333, A 0.000, B 0.000, C 0.000 }
gfCNCPoint3[2763] = {X 29.6250, Y 21.7366, Z -3.8333, A 0.000, B 0.000, C 0.000 }
gfCNCPoint3[2764] = {X 29.5123, Y 23.4559, Z -3.8333, A 0.000, B 0.000, C 0.000 }
gfCNCPoint3[2765] = {X 29.2033, Y 25.1510, Z -3.8333, A 0.000, B 0.000, C 0.000 }
gfCNCPoint3[2766] = {X 28.7611, Y 26.5972, Z -3.8333, A 0.000, B 0.000, C 0.000 }
gfCNCPoint3[2767] = {X 28.1360, Y 27.9742, Z -3.8333, A 0.000, B 0.000, C 0.000 }
gfCNCPoint3[2768] = {X 27.3382, Y 29.2590, Z -3.8333, A 0.000, B 0.000, C 0.000 }
gfCNCPoint3[2769] = {X 26.3813, Y 30.4300, Z -3.8333, A 0.000, B 0.000, C 0.000 }
gfCNCPoint3[2770] = {X 25.2812, Y 31.4677, Z -3.8333, A 0.000, B 0.000, C 0.000 }
gfCNCPoint3[2771] = {X 26.0852, Y 31.8098, Z -3.8333, A 0.000, B 0.000, C 0.000 }
gfCNCPoint3[2772] = {X 26.8039, Y 32.3067, Z -3.8333, A 0.000, B 0.000, C 0.000 }
gfCNCPoint3[2773] = {X 27.4080, Y 32.9381, Z -3.8333, A 0.000, B 0.000, C 0.000 }
gfCNCPoint3[2774] = {X 27.8726, Y 33.6781, Z -3.8333, A 0.000, B 0.000, C 0.000 }
gfCNCPoint3[2775] = {X 30.9100, Y 39.9530, Z -3.8333, A 0.000, B 0.000, C 0.000 }
gfCNCPoint3[2776] = {X 31.2306, Y 40.8622, Z -3.8333, A 0.000, B 0.000, C 0.000 }
gfCNCPoint3[2777] = {X 31.3415, Y 41.8197, Z -3.8333, A 0.000, B 0.000, C 0.000 }
gfCNCPoint3[2778] = {X 31.2374, Y 42.7781, Z -3.8333, A 0.000, B 0.000, C 0.000 }
gfCNCPoint3[2779] = {X 30.9234, Y 43.6895, Z -3.8333, A 0.000, B 0.000, C 0.000 }
gfCNCPoint3[2780] = {X 30.4150, Y 44.5085, Z -3.8333, A 0.000, B 0.000, C 0.000 }
gfCNCPoint3[2781] = {X 29.7377, Y 45.1945, Z -3.8333, A 0.000, B 0.000, C 0.000 }
gfCNCPoint3[2782] = {X 29.2015, Y 45.6280, Z -3.8333, A 0.000, B 0.000, C 0.000 }
gfCNCPoint3[2783] = {X 28.4971, Y 46.0913, Z -3.8333, A 0.000, B 0.000, C 0.000 }
gfCNCPoint3[2784] = {X 27.7163, Y 46.4095, Z -3.8333, A 0.000, B 0.000, C 0.000 }
gfCNCPoint3[2785] = {X 26.8887, Y 46.5705, Z -3.8333, A 0.000, B 0.000, C 0.000 }
gfCNCPoint3[2786] = {X 26.0455, Y 46.5683, Z -3.8333, A 0.000, B 0.000, C 0.000 }
gfCNCPoint3[2787] = {X 25.2188, Y 46.4030, Z -3.8333, A 0.000, B 0.000, C 0.000 }
gfCNCPoint3[2788] = {X 23.4195, Y 47.3541, Z -3.8333, A 0.000, B 0.000, C 0.000 }
gfCNCPoint3[2789] = {X 21.5579, Y 48.1768, Z -3.8333, A 0.000, B 0.000, C 0.000 }
gfCNCPoint3[2790] = {X 19.6433, Y 48.8670, Z -3.8333, A 0.000, B 0.000, C 0.000 }
gfCNCPoint3[2791] = {X 17.4503, Y 49.4711, Z -3.8333, A 0.000, B 0.000, C 0.000 }
gfCNCPoint3[2792] = {X 15.2081, Y 49.8541, Z -3.8333, A 0.000, B 0.000, C 0.000 }
gfCNCPoint3[2793] = {X 12.9390, Y 50.0123, Z -3.8333, A 0.000, B 0.000, C 0.000 }
gfCNCPoint3[2794] = {X 10.6653, Y 49.9442, Z -3.8333, A 0.000, B 0.000, C 0.000 }
gfCNCPoint3[2795] = {X 8.4097, Y 49.6503, Z -3.8333, A 0.000, B 0.000, C 0.000 }
gfCNCPoint3[2796] = {X 6.5298, Y 49.2150, Z -3.8333, A 0.000, B 0.000, C 0.000 }
gfCNCPoint3[2797] = {X 4.7109, Y 48.5705, Z -3.8333, A 0.000, B 0.000, C 0.000 }
gfCNCPoint3[2798] = {X 2.9762, Y 47.7251, Z -3.8333, A 0.000, B 0.000, C 0.000 }
gfCNCPoint3[2799] = {X 1.3479, Y 46.6896, Z -3.8333, A 0.000, B 0.000, C 0.000 }
gfCNCPoint3[2800] = {X 0.6486, Y 46.1466, Z -3.8333, A 0.000, B 0.000, C 0.000 }
gfCNCPoint3[2801] = {X -0.4847, Y 45.1285, Z -3.8333, A 0.000, B 0.000, C 0.000 }
gfCNCPoint3[2802] = {X -1.4910, Y 43.9848, Z -3.8333, A 0.000, B 0.000, C 0.000 }
gfCNCPoint3[2803] = {X -2.3567, Y 42.7313, Z -3.8333, A 0.000, B 0.000, C 0.000 }
gfCNCPoint3[2804] = {X -3.0697, Y 41.3851, Z -3.8333, A 0.000, B 0.000, C 0.000 }
gfCNCPoint3[2805] = {X -3.6204, Y 39.9647, Z -3.8333, A 0.000, B 0.000, C 0.000 }
gfCNCPoint3[2806] = {X -3.6591, Y 39.8423, Z -3.8333, A 0.000, B 0.000, C 0.000 }
gfCNCPoint3[2807] = {X -3.6965, Y 39.7196, Z -3.8333, A 0.000, B 0.000, C 0.000 }
gfCNCPoint3[2808] = {X -4.8459, Y 35.8883, Z -3.8333, A 0.000, B 0.000, C 0.000 }
gfCNCPoint3[2809] = {X -7.9939, Y 36.0001, Z -3.8333, A 0.000, B 0.000, C 0.000 }
gfCNCPoint3[2810] = {X -7.9939, Y 36.0001, Z -0.8333, A 0.000, B 0.000, C 0.000 }
gfCNCPoint3[2811] = {X -7.9939, Y 36.0001, Z 11.0000, A 0.000, B 0.000, C 0.000 }
gfCNCPoint3[2812] = {X 608.0000, Y 40.1199, Z 11.0000, A 0.000, B 0.000, C 0.000 }
gfCNCPoint3[2813] = {X 608.0000, Y 40.1199, Z -0.8333, A 0.000, B 0.000, C 0.000 }
gfCNCPoint3[2814] = {X 608.0000, Y 40.1199, Z -3.8333, A 0.000, B 0.000, C 0.000 }
gfCNCPoint3[2815] = {X 603.6965, Y 47.2356, Z -3.8333, A 0.000, B 0.000, C 0.000 }
gfCNCPoint3[2816] = {X 603.6633, Y 47.2896, Z -3.8333, A 0.000, B 0.000, C 0.000 }
gfCNCPoint3[2817] = {X 603.6293, Y 47.3431, Z -3.8333, A 0.000, B 0.000, C 0.000 }
gfCNCPoint3[2818] = {X 603.0930, Y 48.0159, Z -3.8333, A 0.000, B 0.000, C 0.000 }
gfCNCPoint3[2819] = {X 602.4339, Y 48.5691, Z -3.8333, A 0.000, B 0.000, C 0.000 }
gfCNCPoint3[2820] = {X 601.6783, Y 48.9807, Z -3.8333, A 0.000, B 0.000, C 0.000 }
gfCNCPoint3[2821] = {X 600.8561, Y 49.2343, Z -3.8333, A 0.000, B 0.000, C 0.000 }
gfCNCPoint3[2822] = {X 600.0000, Y 49.3200, Z -3.8333, A 0.000, B 0.000, C 0.000 }
gfCNCPoint3[2823] = {X 593.5565, Y 49.3200, Z -3.8333, A 0.000, B 0.000, C 0.000 }
gfCNCPoint3[2824] = {X 592.5952, Y 49.2117, Z -3.8333, A 0.000, B 0.000, C 0.000 }
gfCNCPoint3[2825] = {X 591.6822, Y 48.8922, Z -3.8333, A 0.000, B 0.000, C 0.000 }
gfCNCPoint3[2826] = {X 590.8631, Y 48.3775, Z -3.8333, A 0.000, B 0.000, C 0.000 }
gfCNCPoint3[2827] = {X 590.1790, Y 47.6935, Z -3.8333, A 0.000, B 0.000, C 0.000 }
gfCNCPoint3[2828] = {X 589.6643, Y 46.8744, Z -3.8333, A 0.000, B 0.000, C 0.000 }
gfCNCPoint3[2829] = {X 589.3448, Y 45.9613, Z -3.8333, A 0.000, B 0.000, C 0.000 }
gfCNCPoint3[2830] = {X 589.2365, Y 45.0000, Z -3.8333, A 0.000, B 0.000, C 0.000 }
gfCNCPoint3[2831] = {X 589.2365, Y 44.0645, Z -3.8333, A 0.000, B 0.000, C 0.000 }
gfCNCPoint3[2832] = {X 589.3410, Y 43.1363, Z -3.8333, A 0.000, B 0.000, C 0.000 }
gfCNCPoint3[2833] = {X 589.6407, Y 42.2516, Z -3.8333, A 0.000, B 0.000, C 0.000 }
gfCNCPoint3[2834] = {X 590.1219, Y 41.4511, Z -3.8333, A 0.000, B 0.000, C 0.000 }
gfCNCPoint3[2835] = {X 590.7625, Y 40.7713, Z -3.8333, A 0.000, B 0.000, C 0.000 }
gfCNCPoint3[2836] = {X 590.7630, Y 33.5305, Z -3.8333, A 0.000, B 0.000, C 0.000 }
gfCNCPoint3[2837] = {X 585.4453, Y 46.6524, Z -3.8333, A 0.000, B 0.000, C 0.000 }
gfCNCPoint3[2838] = {X 585.0755, Y 47.3550, Z -3.8333, A 0.000, B 0.000, C 0.000 }
gfCNCPoint3[2839] = {X 584.5834, Y 47.9780, Z -3.8333, A 0.000, B 0.000, C 0.000 }
gfCNCPoint3[2840] = {X 583.9856, Y 48.5004, Z -3.8333, A 0.000, B 0.000, C 0.000 }
gfCNCPoint3[2841] = {X 583.3023, Y 48.9046, Z -3.8333, A 0.000, B 0.000, C 0.000 }
gfCNCPoint3[2842] = {X 582.3585, Y 49.2242, Z -3.8333, A 0.000, B 0.000, C 0.000 }
gfCNCPoint3[2843] = {X 581.3666, Y 49.3191, Z -3.8333, A 0.000, B 0.000, C 0.000 }
gfCNCPoint3[2844] = {X 580.3794, Y 49.1842, Z -3.8333, A 0.000, B 0.000, C 0.000 }
gfCNCPoint3[2845] = {X 579.4493, Y 48.8268, Z -3.8333, A 0.000, B 0.000, C 0.000 }
gfCNCPoint3[2846] = {X 578.6259, Y 48.2657, Z -3.8333, A 0.000, B 0.000, C 0.000 }
gfCNCPoint3[2847] = {X 577.9529, Y 47.5309, Z -3.8333, A 0.000, B 0.000, C 0.000 }
gfCNCPoint3[2848] = {X 577.4662, Y 46.6615, Z -3.8333, A 0.000, B 0.000, C 0.000 }
gfCNCPoint3[2849] = {X 572.0186, Y 33.3407, Z -3.8333, A 0.000, B 0.000, C 0.000 }
gfCNCPoint3[2850] = {X 572.0189, Y 40.7699, Z -3.8333, A 0.000, B 0.000, C 0.000 }
gfCNCPoint3[2851] = {X 572.6574, Y 41.4410, Z -3.8333, A 0.000, B 0.000, C 0.000 }
gfCNCPoint3[2852] = {X 573.1381, Y 42.2327, Z -3.8333, A 0.000, B 0.000, C 0.000 }
gfCNCPoint3[2853] = {X 573.4390, Y 43.1087, Z -3.8333, A 0.000, B 0.000, C 0.000 }
gfCNCPoint3[2854] = {X 573.5463, Y 44.0287, Z -3.8333, A 0.000, B 0.000, C 0.000 }
gfCNCPoint3[2855] = {X 573.5464, Y 45.0000, Z -3.8333, A 0.000, B 0.000, C 0.000 }
gfCNCPoint3[2856] = {X 573.4381, Y 45.9613, Z -3.8333, A 0.000, B 0.000, C 0.000 }
gfCNCPoint3[2857] = {X 573.1186, Y 46.8744, Z -3.8333, A 0.000, B 0.000, C 0.000 }
gfCNCPoint3[2858] = {X 572.6039, Y 47.6935, Z -3.8333, A 0.000, B 0.000, C 0.000 }
gfCNCPoint3[2859] = {X 571.9199, Y 48.3775, Z -3.8333, A 0.000, B 0.000, C 0.000 }
gfCNCPoint3[2860] = {X 571.1008, Y 48.8922, Z -3.8333, A 0.000, B 0.000, C 0.000 }
gfCNCPoint3[2861] = {X 570.1877, Y 49.2117, Z -3.8333, A 0.000, B 0.000, C 0.000 }
gfCNCPoint3[2862] = {X 569.2264, Y 49.3200, Z -3.8333, A 0.000, B 0.000, C 0.000 }
gfCNCPoint3[2863] = {X 562.4443, Y 49.3200, Z -3.8333, A 0.000, B 0.000, C 0.000 }
gfCNCPoint3[2864] = {X 561.4830, Y 49.2117, Z -3.8333, A 0.000, B 0.000, C 0.000 }
gfCNCPoint3[2865] = {X 560.5699, Y 48.8922, Z -3.8333, A 0.000, B 0.000, C 0.000 }
gfCNCPoint3[2866] = {X 559.7508, Y 48.3775, Z -3.8333, A 0.000, B 0.000, C 0.000 }
gfCNCPoint3[2867] = {X 559.0668, Y 47.6935, Z -3.8333, A 0.000, B 0.000, C 0.000 }
gfCNCPoint3[2868] = {X 558.5521, Y 46.8744, Z -3.8333, A 0.000, B 0.000, C 0.000 }
gfCNCPoint3[2869] = {X 558.2326, Y 45.9613, Z -3.8333, A 0.000, B 0.000, C 0.000 }
gfCNCPoint3[2870] = {X 558.1243, Y 45.0000, Z -3.8333, A 0.000, B 0.000, C 0.000 }
gfCNCPoint3[2871] = {X 558.1243, Y 44.0646, Z -3.8333, A 0.000, B 0.000, C 0.000 }
gfCNCPoint3[2872] = {X 558.2286, Y 43.1360, Z -3.8333, A 0.000, B 0.000, C 0.000 }
gfCNCPoint3[2873] = {X 558.5286, Y 42.2510, Z -3.8333, A 0.000, B 0.000, C 0.000 }
gfCNCPoint3[2874] = {X 559.0105, Y 41.4504, Z -3.8333, A 0.000, B 0.000, C 0.000 }
gfCNCPoint3[2875] = {X 559.6521, Y 40.7710, Z -3.8333, A 0.000, B 0.000, C 0.000 }
gfCNCPoint3[2876] = {X 559.6521, Y 9.2304, Z -3.8333, A 0.000, B 0.000, C 0.000 }
gfCNCPoint3[2877] = {X 559.0136, Y 8.5594, Z -3.8333, A 0.000, B 0.000, C 0.000 }
gfCNCPoint3[2878] = {X 558.5328, Y 7.7678, Z -3.8333, A 0.000, B 0.000, C 0.000 }
gfCNCPoint3[2879] = {X 558.2318, Y 6.8918, Z -3.8333, A 0.000, B 0.000, C 0.000 }
gfCNCPoint3[2880] = {X 558.1245, Y 5.9718, Z -3.8333, A 0.000, B 0.000, C 0.000 }
gfCNCPoint3[2881] = {X 558.1243, Y 5.0000, Z -3.8333, A 0.000, B 0.000, C 0.000 }
gfCNCPoint3[2882] = {X 558.2326, Y 4.0387, Z -3.8333, A 0.000, B 0.000, C 0.000 }
gfCNCPoint3[2883] = {X 558.5521, Y 3.1256, Z -3.8333, A 0.000, B 0.000, C 0.000 }
gfCNCPoint3[2884] = {X 559.0668, Y 2.3065, Z -3.8333, A 0.000, B 0.000, C 0.000 }
gfCNCPoint3[2885] = {X 559.7508, Y 1.6225, Z -3.8333, A 0.000, B 0.000, C 0.000 }
gfCNCPoint3[2886] = {X 560.5699, Y 1.1078, Z -3.8333, A 0.000, B 0.000, C 0.000 }
gfCNCPoint3[2887] = {X 561.4830, Y 0.7883, Z -3.8333, A 0.000, B 0.000, C 0.000 }
gfCNCPoint3[2888] = {X 562.4443, Y 0.6800, Z -3.8333, A 0.000, B 0.000, C 0.000 }
gfCNCPoint3[2889] = {X 570.9376, Y 0.6800, Z -3.8333, A 0.000, B 0.000, C 0.000 }
gfCNCPoint3[2890] = {X 571.8988, Y 0.7883, Z -3.8333, A 0.000, B 0.000, C 0.000 }
gfCNCPoint3[2891] = {X 572.8119, Y 1.1078, Z -3.8333, A 0.000, B 0.000, C 0.000 }
gfCNCPoint3[2892] = {X 573.6310, Y 1.6225, Z -3.8333, A 0.000, B 0.000, C 0.000 }
gfCNCPoint3[2893] = {X 574.3151, Y 2.3065, Z -3.8333, A 0.000, B 0.000, C 0.000 }
gfCNCPoint3[2894] = {X 574.8297, Y 3.1256, Z -3.8333, A 0.000, B 0.000, C 0.000 }
gfCNCPoint3[2895] = {X 575.1492, Y 4.0387, Z -3.8333, A 0.000, B 0.000, C 0.000 }
gfCNCPoint3[2896] = {X 575.2576, Y 5.0000, Z -3.8333, A 0.000, B 0.000, C 0.000 }
gfCNCPoint3[2897] = {X 575.2576, Y 5.9342, Z -3.8333, A 0.000, B 0.000, C 0.000 }
gfCNCPoint3[2898] = {X 575.1835, Y 6.7306, Z -3.8333, A 0.000, B 0.000, C 0.000 }
gfCNCPoint3[2899] = {X 574.9638, Y 7.4998, Z -3.8333, A 0.000, B 0.000, C 0.000 }
gfCNCPoint3[2900] = {X 574.6062, Y 8.2152, Z -3.8333, A 0.000, B 0.000, C 0.000 }
gfCNCPoint3[2901] = {X 581.1909, Y 24.3702, Z -3.8333, A 0.000, B 0.000, C 0.000 }
gfCNCPoint3[2902] = {X 587.8458, Y 8.0943, Z -3.8333, A 0.000, B 0.000, C 0.000 }
gfCNCPoint3[2903] = {X 587.5317, Y 7.4231, Z -3.8333, A 0.000, B 0.000, C 0.000 }
gfCNCPoint3[2904] = {X 587.3369, Y 6.7082, Z -3.8333, A 0.000, B 0.000, C 0.000 }
gfCNCPoint3[2905] = {X 587.2671, Y 5.9705, Z -3.8333, A 0.000, B 0.000, C 0.000 }
gfCNCPoint3[2906] = {X 587.2670, Y 5.0000, Z -3.8333, A 0.000, B 0.000, C 0.000 }
gfCNCPoint3[2907] = {X 587.3753, Y 4.0387, Z -3.8333, A 0.000, B 0.000, C 0.000 }
gfCNCPoint3[2908] = {X 587.6948, Y 3.1256, Z -3.8333, A 0.000, B 0.000, C 0.000 }
gfCNCPoint3[2909] = {X 588.2094, Y 2.3065, Z -3.8333, A 0.000, B 0.000, C 0.000 }
gfCNCPoint3[2910] = {X 588.8935, Y 1.6225, Z -3.8333, A 0.000, B 0.000, C 0.000 }
gfCNCPoint3[2911] = {X 589.7126, Y 1.1078, Z -3.8333, A 0.000, B 0.000, C 0.000 }
gfCNCPoint3[2912] = {X 590.6257, Y 0.7883, Z -3.8333, A 0.000, B 0.000, C 0.000 }
gfCNCPoint3[2913] = {X 591.5870, Y 0.6800, Z -3.8333, A 0.000, B 0.000, C 0.000 }
gfCNCPoint3[2914] = {X 600.0000, Y 0.6800, Z -3.8333, A 0.000, B 0.000, C 0.000 }
gfCNCPoint3[2915] = {X 600.8561, Y 0.7657, Z -3.8333, A 0.000, B 0.000, C 0.000 }
gfCNCPoint3[2916] = {X 601.6783, Y 1.0193, Z -3.8333, A 0.000, B 0.000, C 0.000 }
gfCNCPoint3[2917] = {X 602.4339, Y 1.4309, Z -3.8333, A 0.000, B 0.000, C 0.000 }
gfCNCPoint3[2918] = {X 603.0930, Y 1.9841, Z -3.8333, A 0.000, B 0.000, C 0.000 }
gfCNCPoint3[2919] = {X 603.6293, Y 2.6569, Z -3.8333, A 0.000, B 0.000, C 0.000 }
gfCNCPoint3[2920] = {X 603.6633, Y 2.7104, Z -3.8333, A 0.000, B 0.000, C 0.000 }
gfCNCPoint3[2921] = {X 603.6965, Y 2.7644, Z -3.8333, A 0.000, B 0.000, C 0.000 }
gfCNCPoint3[2922] = {X 608.0000, Y 9.8801, Z -3.8333, A 0.000, B 0.000, C 0.000 }
gfCNCPoint3[2923] = {X 608.0000, Y 9.8801, Z -0.8333, A 0.000, B 0.000, C 0.000 }
gfCNCPoint3[2924] = {X 608.0000, Y 9.8801, Z 11.0000, A 0.000, B 0.000, C 0.000 }
gfCNCPoint3[2925] = {X -7.6965, Y 16.7864, Z 11.0000, A 0.000, B 0.000, C 0.000 }
gfCNCPoint3[2926] = {X -7.6965, Y 16.7864, Z -0.8333, A 0.000, B 0.000, C 0.000 }
gfCNCPoint3[2927] = {X -7.6965, Y 16.7864, Z -3.8333, A 0.000, B 0.000, C 0.000 }
gfCNCPoint3[2928] = {X -4.6245, Y 16.7864, Z -3.8333, A 0.000, B 0.000, C 0.000 }
gfCNCPoint3[2929] = {X -3.6965, Y 12.8955, Z -3.8333, A 0.000, B 0.000, C 0.000 }
gfCNCPoint3[2930] = {X -3.6291, Y 12.6464, Z -3.8333, A 0.000, B 0.000, C 0.000 }
gfCNCPoint3[2931] = {X -3.5466, Y 12.4019, Z -3.8333, A 0.000, B 0.000, C 0.000 }
gfCNCPoint3[2932] = {X -3.1001, Y 11.5271, Z -3.8333, A 0.000, B 0.000, C 0.000 }
gfCNCPoint3[2933] = {X -2.4643, Y 10.7785, Z -3.8333, A 0.000, B 0.000, C 0.000 }
gfCNCPoint3[2934] = {X -1.6733, Y 10.1963, Z -3.8333, A 0.000, B 0.000, C 0.000 }
gfCNCPoint3[2935] = {X -1.0760, Y 9.8556, Z -3.8333, A 0.000, B 0.000, C 0.000 }
gfCNCPoint3[2936] = {X -0.1977, Y 9.4785, Z -3.8333, A 0.000, B 0.000, C 0.000 }
gfCNCPoint3[2937] = {X 0.7428, Y 9.3079, Z -3.8333, A 0.000, B 0.000, C 0.000 }
gfCNCPoint3[2938] = {X 1.6977, Y 9.3522, Z -3.8333, A 0.000, B 0.000, C 0.000 }
gfCNCPoint3[2939] = {X 2.6183, Y 9.6093, Z -3.8333, A 0.000, B 0.000, C 0.000 }
gfCNCPoint3[2940] = {X 3.4093, Y 9.2342, Z -3.8333, A 0.000, B 0.000, C 0.000 }
gfCNCPoint3[2941] = {X 4.2257, Y 8.9185, Z -3.8333, A 0.000, B 0.000, C 0.000 }
gfCNCPoint3[2942] = {X 6.1302, Y 8.2519, Z -3.8333, A 0.000, B 0.000, C 0.000 }
gfCNCPoint3[2943] = {X 8.0851, Y 7.7520, Z -3.8333, A 0.000, B 0.000, C 0.000 }
gfCNCPoint3[2944] = {X 10.0758, Y 7.4226, Z -3.8333, A 0.000, B 0.000, C 0.000 }
gfCNCPoint3[2945] = {X 12.0875, Y 7.2661, Z -3.8333, A 0.000, B 0.000, C 0.000 }
gfCNCPoint3[2946] = {X 14.1052, Y 7.2836, Z -3.8333, A 0.000, B 0.000, C 0.000 }
gfCNCPoint3[2947] = {X 16.1139, Y 7.4751, Z -3.8333, A 0.000, B 0.000, C 0.000 }
gfCNCPoint3[2948] = {X 17.9288, Y 7.8071, Z -3.8333, A 0.000, B 0.000, C 0.000 }
gfCNCPoint3[2949] = {X 19.6982, Y 8.3298, Z -3.8333, A 0.000, B 0.000, C 0.000 }
gfCNCPoint3[2950] = {X 21.4023, Y 9.0371, Z -3.8333, A 0.000, B 0.000, C 0.000 }
gfCNCPoint3[2951] = {X 23.0218, Y 9.9211, Z -3.8333, A 0.000, B 0.000, C 0.000 }
gfCNCPoint3[2952] = {X 24.5383, Y 10.9719, Z -3.8333, A 0.000, B 0.000, C 0.000 }
gfCNCPoint3[2953] = {X 25.6168, Y 11.9148, Z -3.8333, A 0.000, B 0.000, C 0.000 }
gfCNCPoint3[2954] = {X 26.5843, Y 12.9714, Z -3.8333, A 0.000, B 0.000, C 0.000 }
gfCNCPoint3[2955] = {X 27.4287, Y 14.1287, Z -3.8333, A 0.000, B 0.000, C 0.000 }
gfCNCPoint3[2956] = {X 28.1398, Y 15.3723, Z -3.8333, A 0.000, B 0.000, C 0.000 }
gfCNCPoint3[2957] = {X 28.7088, Y 16.6870, Z -3.8333, A 0.000, B 0.000, C 0.000 }
gfCNCPoint3[2958] = {X 29.1806, Y 18.3344, Z -3.8333, A 0.000, B 0.000, C 0.000 }
gfCNCPoint3[2959] = {X 29.4606, Y 20.0250, Z -3.8333, A 0.000, B 0.000, C 0.000 }
gfCNCPoint3[2960] = {X 29.5450, Y 21.7366, Z -3.8333, A 0.000, B 0.000, C 0.000 }
gfCNCPoint3[2961] = {X 29.4329, Y 23.4465, Z -3.8333, A 0.000, B 0.000, C 0.000 }
gfCNCPoint3[2962] = {X 29.1255, Y 25.1324, Z -3.8333, A 0.000, B 0.000, C 0.000 }
gfCNCPoint3[2963] = {X 28.6756, Y 26.5971, Z -3.8333, A 0.000, B 0.000, C 0.000 }
gfCNCPoint3[2964] = {X 28.0367, Y 27.9898, Z -3.8333, A 0.000, B 0.000, C 0.000 }
gfCNCPoint3[2965] = {X 27.2200, Y 29.2862, Z -3.8333, A 0.000, B 0.000, C 0.000 }
gfCNCPoint3[2966] = {X 26.2397, Y 30.4637, Z -3.8333, A 0.000, B 0.000, C 0.000 }
gfCNCPoint3[2967] = {X 25.1128, Y 31.5019, Z -3.8333, A 0.000, B 0.000, C 0.000 }
gfCNCPoint3[2968] = {X 25.2523, Y 31.5425, Z -3.8333, A 0.000, B 0.000, C 0.000 }
gfCNCPoint3[2969] = {X 25.3904, Y 31.5877, Z -3.8333, A 0.000, B 0.000, C 0.000 }
gfCNCPoint3[2970] = {X 26.1379, Y 31.9316, Z -3.8333, A 0.000, B 0.000, C 0.000 }
gfCNCPoint3[2971] = {X 26.8049, Y 32.4134, Z -3.8333, A 0.000, B 0.000, C 0.000 }
gfCNCPoint3[2972] = {X 27.3662, Y 33.0150, Z -3.8333, A 0.000, B 0.000, C 0.000 }
gfCNCPoint3[2973] = {X 27.8009, Y 33.7136, Z -3.8333, A 0.000, B 0.000, C 0.000 }
gfCNCPoint3[2974] = {X 30.8380, Y 39.9879, Z -3.8333, A 0.000, B 0.000, C 0.000 }
gfCNCPoint3[2975] = {X 31.1526, Y 40.8802, Z -3.8333, A 0.000, B 0.000, C 0.000 }
gfCNCPoint3[2976] = {X 31.2615, Y 41.8200, Z -3.8333, A 0.000, B 0.000, C 0.000 }
gfCNCPoint3[2977] = {X 31.1593, Y 42.7606, Z -3.8333, A 0.000, B 0.000, C 0.000 }
gfCNCPoint3[2978] = {X 30.8511, Y 43.6551, Z -3.8333, A 0.000, B 0.000, C 0.000 }
gfCNCPoint3[2979] = {X 30.3522, Y 44.4590, Z -3.8333, A 0.000, B 0.000, C 0.000 }
gfCNCPoint3[2980] = {X 29.6874, Y 45.1323, Z -3.8333, A 0.000, B 0.000, C 0.000 }
gfCNCPoint3[2981] = {X 29.1512, Y 45.5658, Z -3.8333, A 0.000, B 0.000, C 0.000 }
gfCNCPoint3[2982] = {X 28.4537, Y 46.0237, Z -3.8333, A 0.000, B 0.000, C 0.000 }
gfCNCPoint3[2983] = {X 27.6802, Y 46.3368, Z -3.8333, A 0.000, B 0.000, C 0.000 }
gfCNCPoint3[2984] = {X 26.8605, Y 46.4928, Z -3.8333, A 0.000, B 0.000, C 0.000 }
gfCNCPoint3[2985] = {X 26.0261, Y 46.4859, Z -3.8333, A 0.000, B 0.000, C 0.000 }
gfCNCPoint3[2986] = {X 25.2091, Y 46.3163, Z -3.8333, A 0.000, B 0.000, C 0.000 }
gfCNCPoint3[2987] = {X 23.4053, Y 47.2720, Z -3.8333, A 0.000, B 0.000, C 0.000 }
gfCNCPoint3[2988] = {X 21.5387, Y 48.0983, Z -3.8333, A 0.000, B 0.000, C 0.000 }
gfCNCPoint3[2989] = {X 19.6186, Y 48.7909, Z -3.8333, A 0.000, B 0.000, C 0.000 }
gfCNCPoint3[2990] = {X 17.4331, Y 49.3929, Z -3.8333, A 0.000, B 0.000, C 0.000 }
gfCNCPoint3[2991] = {X 15.1987, Y 49.7747, Z -3.8333, A 0.000, B 0.000, C 0.000 }
gfCNCPoint3[2992] = {X 12.9373, Y 49.9324, Z -3.8333, A 0.000, B 0.000, C 0.000 }
gfCNCPoint3[2993] = {X 10.6715, Y 49.8644, Z -3.8333, A 0.000, B 0.000, C 0.000 }
gfCNCPoint3[2994] = {X 8.4237, Y 49.5716, Z -3.8333, A 0.000, B 0.000, C 0.000 }
gfCNCPoint3[2995] = {X 6.5528, Y 49.1384, Z -3.8333, A 0.000, B 0.000, C 0.000 }
gfCNCPoint3[2996] = {X 4.7427, Y 48.4971, Z -3.8333, A 0.000, B 0.000, C 0.000 }
gfCNCPoint3[2997] = {X 3.0163, Y 47.6559, Z -3.8333, A 0.000, B 0.000, C 0.000 }
gfCNCPoint3[2998] = {X 1.3958, Y 46.6255, Z -3.8333, A 0.000, B 0.000, C 0.000 }
gfCNCPoint3[2999] = {X 0.6985, Y 46.0840, Z -3.8333, A 0.000, B 0.000, C 0.000 }
gfCNCPoint3[3000] = {X -0.4278, Y 45.0722, Z -3.8333, A 0.000, B 0.000, C 0.000 }
gfCNCPoint3[3001] = {X -1.4280, Y 43.9356, Z -3.8333, A 0.000, B 0.000, C 0.000 }
gfCNCPoint3[3002] = {X -2.2883, Y 42.6898, Z -3.8333, A 0.000, B 0.000, C 0.000 }
gfCNCPoint3[3003] = {X -2.9970, Y 41.3518, Z -3.8333, A 0.000, B 0.000, C 0.000 }
gfCNCPoint3[3004] = {X -3.5442, Y 39.9402, Z -3.8333, A 0.000, B 0.000, C 0.000 }
gfCNCPoint3[3005] = {X -3.6230, Y 39.6863, Z -3.8333, A 0.000, B 0.000, C 0.000 }
gfCNCPoint3[3006] = {X -3.6965, Y 39.4309, Z -3.8333, A 0.000, B 0.000, C 0.000 }
gfCNCPoint3[3007] = {X -4.7636, Y 35.5759, Z -3.8333, A 0.000, B 0.000, C 0.000 }
gfCNCPoint3[3008] = {X -8.0034, Y 35.6252, Z -3.8333, A 0.000, B 0.000, C 0.000 }
gfCNCPoint3[3009] = {X -8.0034, Y 35.6252, Z -0.8333, A 0.000, B 0.000, C 0.000 }
gfCNCPoint3[3010] = {X -8.0034, Y 35.6252, Z 11.0000, A 0.000, B 0.000, C 0.000 }
gfCNCPoint3[3011] = {X -7.6965, Y 17.3012, Z 11.0000, A 0.000, B 0.000, C 0.000 }
gfCNCPoint3[3012] = {X -7.6965, Y 17.3012, Z -0.8333, A 0.000, B 0.000, C 0.000 }
gfCNCPoint3[3013] = {X -7.6965, Y 17.3012, Z -3.8333, A 0.000, B 0.000, C 0.000 }
gfCNCPoint3[3014] = {X -4.2193, Y 17.3012, Z -3.8333, A 0.000, B 0.000, C 0.000 }
gfCNCPoint3[3015] = {X -3.6965, Y 13.3355, Z -3.8333, A 0.000, B 0.000, C 0.000 }
gfCNCPoint3[3016] = {X -3.6095, Y 12.8763, Z -3.8333, A 0.000, B 0.000, C 0.000 }
gfCNCPoint3[3017] = {X -3.4716, Y 12.4298, Z -3.8333, A 0.000, B 0.000, C 0.000 }
gfCNCPoint3[3018] = {X -3.0335, Y 11.5715, Z -3.8333, A 0.000, B 0.000, C 0.000 }
gfCNCPoint3[3019] = {X -2.4097, Y 10.8370, Z -3.8333, A 0.000, B 0.000, C 0.000 }
gfCNCPoint3[3020] = {X -1.6337, Y 10.2658, Z -3.8333, A 0.000, B 0.000, C 0.000 }
gfCNCPoint3[3021] = {X -1.0364, Y 9.9251, Z -3.8333, A 0.000, B 0.000, C 0.000 }
gfCNCPoint3[3022] = {X -0.1658, Y 9.5525, Z -3.8333, A 0.000, B 0.000, C 0.000 }
gfCNCPoint3[3023] = {X 0.7666, Y 9.3865, Z -3.8333, A 0.000, B 0.000, C 0.000 }
gfCNCPoint3[3024] = {X 1.7123, Y 9.4356, Z -3.8333, A 0.000, B 0.000, C 0.000 }
gfCNCPoint3[3025] = {X 2.6224, Y 9.6974, Z -3.8333, A 0.000, B 0.000, C 0.000 }
gfCNCPoint3[3026] = {X 3.4247, Y 9.3147, Z -3.8333, A 0.000, B 0.000, C 0.000 }
gfCNCPoint3[3027] = {X 4.2536, Y 8.9935, Z -3.8333, A 0.000, B 0.000, C 0.000 }
gfCNCPoint3[3028] = {X 6.1519, Y 8.3289, Z -3.8333, A 0.000, B 0.000, C 0.000 }
gfCNCPoint3[3029] = {X 8.1004, Y 7.8306, Z -3.8333, A 0.000, B 0.000, C 0.000 }
gfCNCPoint3[3030] = {X 10.0847, Y 7.5021, Z -3.8333, A 0.000, B 0.000, C 0.000 }
gfCNCPoint3[3031] = {X 12.0899, Y 7.3460, Z -3.8333, A 0.000, B 0.000, C 0.000 }
gfCNCPoint3[3032] = {X 14.1010, Y 7.3635, Z -3.8333, A 0.000, B 0.000, C 0.000 }
gfCNCPoint3[3033] = {X 16.1032, Y 7.5544, Z -3.8333, A 0.000, B 0.000, C 0.000 }
gfCNCPoint3[3034] = {X 17.9099, Y 7.8849, Z -3.8333, A 0.000, B 0.000, C 0.000 }
gfCNCPoint3[3035] = {X 19.6713, Y 8.4051, Z -3.8333, A 0.000, B 0.000, C 0.000 }
gfCNCPoint3[3036] = {X 21.3676, Y 9.1092, Z -3.8333, A 0.000, B 0.000, C 0.000 }
gfCNCPoint3[3037] = {X 22.9797, Y 9.9892, Z -3.8333, A 0.000, B 0.000, C 0.000 }
gfCNCPoint3[3038] = {X 24.4894, Y 11.0352, Z -3.8333, A 0.000, B 0.000, C 0.000 }
gfCNCPoint3[3039] = {X 25.5611, Y 11.9722, Z -3.8333, A 0.000, B 0.000, C 0.000 }
gfCNCPoint3[3040] = {X 26.5225, Y 13.0222, Z -3.8333, A 0.000, B 0.000, C 0.000 }
gfCNCPoint3[3041] = {X 27.3617, Y 14.1723, Z -3.8333, A 0.000, B 0.000, C 0.000 }
gfCNCPoint3[3042] = {X 28.0683, Y 15.4081, Z -3.8333, A 0.000, B 0.000, C 0.000 }
gfCNCPoint3[3043] = {X 28.6337, Y 16.7147, Z -3.8333, A 0.000, B 0.000, C 0.000 }
gfCNCPoint3[3044] = {X 29.1028, Y 18.3531, Z -3.8333, A 0.000, B 0.000, C 0.000 }
gfCNCPoint3[3045] = {X 29.3811, Y 20.0344, Z -3.8333, A 0.000, B 0.000, C 0.000 }
gfCNCPoint3[3046] = {X 29.4650, Y 21.7366, Z -3.8333, A 0.000, B 0.000, C 0.000 }
gfCNCPoint3[3047] = {X 29.3534, Y 23.4372, Z -3.8333, A 0.000, B 0.000, C 0.000 }
gfCNCPoint3[3048] = {X 29.0477, Y 25.1138, Z -3.8333, A 0.000, B 0.000, C 0.000 }
gfCNCPoint3[3049] = {X 28.5894, Y 26.5986, Z -3.8333, A 0.000, B 0.000, C 0.000 }
gfCNCPoint3[3050] = {X 27.9356, Y 28.0082, Z -3.8333, A 0.000, B 0.000, C 0.000 }
gfCNCPoint3[3051] = {X 27.0981, Y 29.3172, Z -3.8333, A 0.000, B 0.000, C 0.000 }
gfCNCPoint3[3052] = {X 26.0923, Y 30.5016, Z -3.8333, A 0.000, B 0.000, C 0.000 }
gfCNCPoint3[3053] = {X 24.9363, Y 31.5401, Z -3.8333, A 0.000, B 0.000, C 0.000 }
gfCNCPoint3[3054] = {X 25.1519, Y 31.5960, Z -3.8333, A 0.000, B 0.000, C 0.000 }
gfCNCPoint3[3055] = {X 25.3642, Y 31.6633, Z -3.8333, A 0.000, B 0.000, C 0.000 }
gfCNCPoint3[3056] = {X 26.0975, Y 32.0007, Z -3.8333, A 0.000, B 0.000, C 0.000 }
gfCNCPoint3[3057] = {X 26.7519, Y 32.4734, Z -3.8333, A 0.000, B 0.000, C 0.000 }
gfCNCPoint3[3058] = {X 27.3027, Y 33.0636, Z -3.8333, A 0.000, B 0.000, C 0.000 }
gfCNCPoint3[3059] = {X 27.7292, Y 33.7491, Z -3.8333, A 0.000, B 0.000, C 0.000 }
gfCNCPoint3[3060] = {X 30.7660, Y 40.0227, Z -3.8333, A 0.000, B 0.000, C 0.000 }
gfCNCPoint3[3061] = {X 31.0747, Y 40.8982, Z -3.8333, A 0.000, B 0.000, C 0.000 }
gfCNCPoint3[3062] = {X 31.1815, Y 41.8203, Z -3.8333, A 0.000, B 0.000, C 0.000 }
gfCNCPoint3[3063] = {X 31.0813, Y 42.7431, Z -3.8333, A 0.000, B 0.000, C 0.000 }
gfCNCPoint3[3064] = {X 30.7789, Y 43.6208, Z -3.8333, A 0.000, B 0.000, C 0.000 }
gfCNCPoint3[3065] = {X 30.2893, Y 44.4095, Z -3.8333, A 0.000, B 0.000, C 0.000 }
gfCNCPoint3[3066] = {X 29.6371, Y 45.0700, Z -3.8333, A 0.000, B 0.000, C 0.000 }
gfCNCPoint3[3067] = {X 29.1010, Y 45.5035, Z -3.8333, A 0.000, B 0.000, C 0.000 }
gfCNCPoint3[3068] = {X 28.4104, Y 45.9561, Z -3.8333, A 0.000, B 0.000, C 0.000 }
gfCNCPoint3[3069] = {X 27.6442, Y 46.2639, Z -3.8333, A 0.000, B 0.000, C 0.000 }
gfCNCPoint3[3070] = {X 26.8324, Y 46.4150, Z -3.8333, A 0.000, B 0.000, C 0.000 }
gfCNCPoint3[3071] = {X 26.0068, Y 46.4033, Z -3.8333, A 0.000, B 0.000, C 0.000 }
gfCNCPoint3[3072] = {X 25.1996, Y 46.2294, Z -3.8333, A 0.000, B 0.000, C 0.000 }
gfCNCPoint3[3073] = {X 23.3914, Y 47.1899, Z -3.8333, A 0.000, B 0.000, C 0.000 }
gfCNCPoint3[3074] = {X 21.5197, Y 48.0198, Z -3.8333, A 0.000, B 0.000, C 0.000 }
gfCNCPoint3[3075] = {X 19.5938, Y 48.7149, Z -3.8333, A 0.000, B 0.000, C 0.000 }
gfCNCPoint3[3076] = {X 17.4159, Y 49.3148, Z -3.8333, A 0.000, B 0.000, C 0.000 }
gfCNCPoint3[3077] = {X 15.1892, Y 49.6952, Z -3.8333, A 0.000, B 0.000, C 0.000 }
gfCNCPoint3[3078] = {X 12.9357, Y 49.8524, Z -3.8333, A 0.000, B 0.000, C 0.000 }
gfCNCPoint3[3079] = {X 10.6777, Y 49.7847, Z -3.8333, A 0.000, B 0.000, C 0.000 }
gfCNCPoint3[3080] = {X 8.4377, Y 49.4928, Z -3.8333, A 0.000, B 0.000, C 0.000 }
gfCNCPoint3[3081] = {X 6.5758, Y 49.0618, Z -3.8333, A 0.000, B 0.000, C 0.000 }
gfCNCPoint3[3082] = {X 4.7744, Y 48.4237, Z -3.8333, A 0.000, B 0.000, C 0.000 }
gfCNCPoint3[3083] = {X 3.0564, Y 47.5867, Z -3.8333, A 0.000, B 0.000, C 0.000 }
gfCNCPoint3[3084] = {X 1.4437, Y 46.5614, Z -3.8333, A 0.000, B 0.000, C 0.000 }
gfCNCPoint3[3085] = {X 0.7480, Y 46.0212, Z -3.8333, A 0.000, B 0.000, C 0.000 }
gfCNCPoint3[3086] = {X -0.3712, Y 45.0157, Z -3.8333, A 0.000, B 0.000, C 0.000 }
gfCNCPoint3[3087] = {X -1.3651, Y 43.8861, Z -3.8333, A 0.000, B 0.000, C 0.000 }
gfCNCPoint3[3088] = {X -2.2200, Y 42.6481, Z -3.8333, A 0.000, B 0.000, C 0.000 }
gfCNCPoint3[3089] = {X -2.9243, Y 41.3185, Z -3.8333, A 0.000, B 0.000, C 0.000 }
gfCNCPoint3[3090] = {X -3.4681, Y 39.9157, Z -3.8333, A 0.000, B 0.000, C 0.000 }
gfCNCPoint3[3091] = {X -3.5888, Y 39.5186, Z -3.8333, A 0.000, B 0.000, C 0.000 }
gfCNCPoint3[3092] = {X -3.6965, Y 39.1177, Z -3.8333, A 0.000, B 0.000, C 0.000 }
gfCNCPoint3[3093] = {X -4.6727, Y 35.2387, Z -3.8333, A 0.000, B 0.000, C 0.000 }
gfCNCPoint3[3094] = {X -8.0051, Y 35.2156, Z -3.8333, A 0.000, B 0.000, C 0.000 }
gfCNCPoint3[3095] = {X -8.0051, Y 35.2156, Z -0.8333, A 0.000, B 0.000, C 0.000 }
gfCNCPoint3[3096] = {X -8.0051, Y 35.2156, Z 11.0000, A 0.000, B 0.000, C 0.000 }
gfCNCPoint3[3097] = {X -7.9979, Y 34.8120, Z 11.0000, A 0.000, B 0.000, C 0.000 }
gfCNCPoint3[3098] = {X -7.9979, Y 34.8120, Z -0.8333, A 0.000, B 0.000, C 0.000 }
gfCNCPoint3[3099] = {X -7.9979, Y 34.8120, Z -3.8333, A 0.000, B 0.000, C 0.000 }
gfCNCPoint3[3100] = {X -4.8496, Y 34.9025, Z -3.8333, A 0.000, B 0.000, C 0.000 }
gfCNCPoint3[3101] = {X -3.6965, Y 31.0723, Z -3.8333, A 0.000, B 0.000, C 0.000 }
gfCNCPoint3[3102] = {X -3.6590, Y 30.9495, Z -3.8333, A 0.000, B 0.000, C 0.000 }
gfCNCPoint3[3103] = {X -3.6204, Y 30.8270, Z -3.8333, A 0.000, B 0.000, C 0.000 }
gfCNCPoint3[3104] = {X -3.4454, Y 30.3131, Z -3.8333, A 0.000, B 0.000, C 0.000 }
gfCNCPoint3[3105] = {X -3.2518, Y 29.8059, Z -3.8333, A 0.000, B 0.000, C 0.000 }
gfCNCPoint3[3106] = {X -2.6172, Y 28.4662, Z -3.8333, A 0.000, B 0.000, C 0.000 }
gfCNCPoint3[3107] = {X -1.8056, Y 27.2257, Z -3.8333, A 0.000, B 0.000, C 0.000 }
gfCNCPoint3[3108] = {X -0.8321, Y 26.1078, Z -3.8333, A 0.000, B 0.000, C 0.000 }
gfCNCPoint3[3109] = {X 0.2851, Y 25.1334, Z -3.8333, A 0.000, B 0.000, C 0.000 }
gfCNCPoint3[3110] = {X 1.5248, Y 24.3207, Z -3.8333, A 0.000, B 0.000, C 0.000 }
gfCNCPoint3[3111] = {X 1.4479, Y 24.2910, Z -3.8333, A 0.000, B 0.000, C 0.000 }
gfCNCPoint3[3112] = {X 1.3716, Y 24.2600, Z -3.8333, A 0.000, B 0.000, C 0.000 }
gfCNCPoint3[3113] = {X 0.6327, Y 23.8625, Z -3.8333, A 0.000, B 0.000, C 0.000 }
gfCNCPoint3[3114] = {X -0.0155, Y 23.3296, Z -3.8333, A 0.000, B 0.000, C 0.000 }
gfCNCPoint3[3115] = {X -0.5484, Y 22.6816, Z -3.8333, A 0.000, B 0.000, C 0.000 }
gfCNCPoint3[3116] = {X -0.9460, Y 21.9427, Z -3.8333, A 0.000, B 0.000, C 0.000 }
gfCNCPoint3[3117] = {X -3.6216, Y 15.3842, Z -3.8333, A 0.000, B 0.000, C 0.000 }
gfCNCPoint3[3118] = {X -3.6605, Y 15.2749, Z -3.8333, A 0.000, B 0.000, C 0.000 }
gfCNCPoint3[3119] = {X -3.6965, Y 15.1645, Z -3.8333, A 0.000, B 0.000, C 0.000 }
gfCNCPoint3[3120] = {X -4.8868, Y 11.3457, Z -3.8333, A 0.000, B 0.000, C 0.000 }
gfCNCPoint3[3121] = {X -7.6965, Y 11.3457, Z -3.8333, A 0.000, B 0.000, C 0.000 }
gfCNCPoint3[3122] = {X -7.6965, Y 11.3457, Z -0.8333, A 0.000, B 0.000, C 0.000 }
gfCNCPoint3[3123] = {X -7.6965, Y 11.3457, Z 11.0000, A 0.000, B 0.000, C 0.000 }
gfCNCPoint3[3124] = {X -8.0048, Y 35.1814, Z 11.0000, A 0.000, B 0.000, C 0.000 }
gfCNCPoint3[3125] = {X -8.0048, Y 35.1814, Z -0.8333, A 0.000, B 0.000, C 0.000 }
gfCNCPoint3[3126] = {X -8.0048, Y 35.1814, Z -3.8333, A 0.000, B 0.000, C 0.000 }
gfCNCPoint3[3127] = {X -4.7782, Y 35.2097, Z -3.8333, A 0.000, B 0.000, C 0.000 }
gfCNCPoint3[3128] = {X -3.6965, Y 31.3587, Z -3.8333, A 0.000, B 0.000, C 0.000 }
gfCNCPoint3[3129] = {X -3.6226, Y 31.1043, Z -3.8333, A 0.000, B 0.000, C 0.000 }
gfCNCPoint3[3130] = {X -3.5442, Y 30.8514, Z -3.8333, A 0.000, B 0.000, C 0.000 }
gfCNCPoint3[3131] = {X -3.3701, Y 30.3400, Z -3.8333, A 0.000, B 0.000, C 0.000 }
gfCNCPoint3[3132] = {X -3.1775, Y 29.8355, Z -3.8333, A 0.000, B 0.000, C 0.000 }
gfCNCPoint3[3133] = {X -2.5301, Y 28.4745, Z -3.8333, A 0.000, B 0.000, C 0.000 }
gfCNCPoint3[3134] = {X -1.6987, Y 27.2175, Z -3.8333, A 0.000, B 0.000, C 0.000 }
gfCNCPoint3[3135] = {X -0.6996, Y 26.0892, Z -3.8333, A 0.000, B 0.000, C 0.000 }
gfCNCPoint3[3136] = {X 0.4476, Y 25.1117, Z -3.8333, A 0.000, B 0.000, C 0.000 }
gfCNCPoint3[3137] = {X 1.7202, Y 24.3044, Z -3.8333, A 0.000, B 0.000, C 0.000 }
gfCNCPoint3[3138] = {X 1.5602, Y 24.2485, Z -3.8333, A 0.000, B 0.000, C 0.000 }
gfCNCPoint3[3139] = {X 1.4025, Y 24.1862, Z -3.8333, A 0.000, B 0.000, C 0.000 }
gfCNCPoint3[3140] = {X 0.6773, Y 23.7960, Z -3.8333, A 0.000, B 0.000, C 0.000 }
gfCNCPoint3[3141] = {X 0.0411, Y 23.2731, Z -3.8333, A 0.000, B 0.000, C 0.000 }
gfCNCPoint3[3142] = {X -0.4819, Y 22.6370, Z -3.8333, A 0.000, B 0.000, C 0.000 }
gfCNCPoint3[3143] = {X -0.8722, Y 21.9118, Z -3.8333, A 0.000, B 0.000, C 0.000 }
gfCNCPoint3[3144] = {X -3.5466, Y 15.3563, Z -3.8333, A 0.000, B 0.000, C 0.000 }
gfCNCPoint3[3145] = {X -3.6291, Y 15.1118, Z -3.8333, A 0.000, B 0.000, C 0.000 }
gfCNCPoint3[3146] = {X -3.6965, Y 14.8627, Z -3.8333, A 0.000, B 0.000, C 0.000 }
gfCNCPoint3[3147] = {X -4.6245, Y 10.9719, Z -3.8333, A 0.000, B 0.000, C 0.000 }
gfCNCPoint3[3148] = {X -7.6965, Y 10.9719, Z -3.8333, A 0.000, B 0.000, C 0.000 }
gfCNCPoint3[3149] = {X -7.6965, Y 10.9719, Z -0.8333, A 0.000, B 0.000, C 0.000 }
gfCNCPoint3[3150] = {X -7.6965, Y 10.9719, Z 11.0000, A 0.000, B 0.000, C 0.000 }
gfCNCPoint3[3151] = {X -8.0040, Y 35.5797, Z 11.0000, A 0.000, B 0.000, C 0.000 }
gfCNCPoint3[3152] = {X -8.0040, Y 35.5797, Z -0.8333, A 0.000, B 0.000, C 0.000 }
gfCNCPoint3[3153] = {X -8.0040, Y 35.5797, Z -3.8333, A 0.000, B 0.000, C 0.000 }
gfCNCPoint3[3154] = {X -4.7003, Y 35.5376, Z -3.8333, A 0.000, B 0.000, C 0.000 }
gfCNCPoint3[3155] = {X -3.6965, Y 31.6656, Z -3.8333, A 0.000, B 0.000, C 0.000 }
gfCNCPoint3[3156] = {X -3.5878, Y 31.2690, Z -3.8333, A 0.000, B 0.000, C 0.000 }
gfCNCPoint3[3157] = {X -3.4680, Y 30.8757, Z -3.8333, A 0.000, B 0.000, C 0.000 }
gfCNCPoint3[3158] = {X -3.2948, Y 30.3670, Z -3.8333, A 0.000, B 0.000, C 0.000 }
gfCNCPoint3[3159] = {X -3.1031, Y 29.8650, Z -3.8333, A 0.000, B 0.000, C 0.000 }
gfCNCPoint3[3160] = {X -2.4414, Y 28.4803, Z -3.8333, A 0.000, B 0.000, C 0.000 }
gfCNCPoint3[3161] = {X -1.5879, Y 27.2049, Z -3.8333, A 0.000, B 0.000, C 0.000 }
gfCNCPoint3[3162] = {X -0.5601, Y 26.0653, Z -3.8333, A 0.000, B 0.000, C 0.000 }
gfCNCPoint3[3163] = {X 0.6206, Y 25.0849, Z -3.8333, A 0.000, B 0.000, C 0.000 }
gfCNCPoint3[3164] = {X 1.9298, Y 24.2841, Z -3.8333, A 0.000, B 0.000, C 0.000 }
gfCNCPoint3[3165] = {X 1.6789, Y 24.2061, Z -3.8333, A 0.000, B 0.000, C 0.000 }
gfCNCPoint3[3166] = {X 1.4334, Y 24.1124, Z -3.8333, A 0.000, B 0.000, C 0.000 }
gfCNCPoint3[3167] = {X 0.7218, Y 23.7296, Z -3.8333, A 0.000, B 0.000, C 0.000 }
gfCNCPoint3[3168] = {X 0.0977, Y 23.2165, Z -3.8333, A 0.000, B 0.000, C 0.000 }
gfCNCPoint3[3169] = {X -0.4155, Y 22.5924, Z -3.8333, A 0.000, B 0.000, C 0.000 }
gfCNCPoint3[3170] = {X -0.7984, Y 21.8809, Z -3.8333, A 0.000, B 0.000, C 0.000 }
gfCNCPoint3[3171] = {X -3.4716, Y 15.3285, Z -3.8333, A 0.000, B 0.000, C 0.000 }
gfCNCPoint3[3172] = {X -3.6095, Y 14.8819, Z -3.8333, A 0.000, B 0.000, C 0.000 }
gfCNCPoint3[3173] = {X -3.6965, Y 14.4227, Z -3.8333, A 0.000, B 0.000, C 0.000 }
gfCNCPoint3[3174] = {X -4.2193, Y 10.4570, Z -3.8333, A 0.000, B 0.000, C 0.000 }
gfCNCPoint3[3175] = {X -7.6965, Y 10.4570, Z -3.8333, A 0.000, B 0.000, C 0.000 }
gfCNCPoint3[3176] = {X -7.6965, Y 10.4570, Z -0.8333, A 0.000, B 0.000, C 0.000 }
gfCNCPoint3[3177] = {X -7.6965, Y 10.4570, Z 11.0000, A 0.000, B 0.000, C 0.000 }
gfCNCPoint3[3178] = {X -7.9934, Y 36.0144, Z 11.0000, A 0.000, B 0.000, C 0.000 }
gfCNCPoint3[3179] = {X -7.9934, Y 36.0144, Z -0.8333, A 0.000, B 0.000, C 0.000 }
gfCNCPoint3[3180] = {X -7.9934, Y 36.0144, Z -3.8333, A 0.000, B 0.000, C 0.000 }
gfCNCPoint3[3181] = {X -4.6145, Y 35.8918, Z -3.8333, A 0.000, B 0.000, C 0.000 }
gfCNCPoint3[3182] = {X -3.6965, Y 31.9986, Z -3.8333, A 0.000, B 0.000, C 0.000 }
gfCNCPoint3[3183] = {X -3.5549, Y 31.4464, Z -3.8333, A 0.000, B 0.000, C 0.000 }
gfCNCPoint3[3184] = {X -3.3918, Y 30.9001, Z -3.8333, A 0.000, B 0.000, C 0.000 }
gfCNCPoint3[3185] = {X -3.2195, Y 30.3940, Z -3.8333, A 0.000, B 0.000, C 0.000 }
gfCNCPoint3[3186] = {X -3.0288, Y 29.8946, Z -3.8333, A 0.000, B 0.000, C 0.000 }
gfCNCPoint3[3187] = {X -2.3507, Y 28.4829, Z -3.8333, A 0.000, B 0.000, C 0.000 }
gfCNCPoint3[3188] = {X -1.4718, Y 27.1867, Z -3.8333, A 0.000, B 0.000, C 0.000 }
gfCNCPoint3[3189] = {X -0.4113, Y 26.0344, Z -3.8333, A 0.000, B 0.000, C 0.000 }
gfCNCPoint3[3190] = {X 0.8077, Y 25.0512, Z -3.8333, A 0.000, B 0.000, C 0.000 }
gfCNCPoint3[3191] = {X 2.1583, Y 24.2585, Z -3.8333, A 0.000, B 0.000, C 0.000 }
gfCNCPoint3[3192] = {X 1.8064, Y 24.1641, Z -3.8333, A 0.000, B 0.000, C 0.000 }
gfCNCPoint3[3193] = {X 1.4643, Y 24.0386, Z -3.8333, A 0.000, B 0.000, C 0.000 }
gfCNCPoint3[3194] = {X 0.7664, Y 23.6632, Z -3.8333, A 0.000, B 0.000, C 0.000 }
gfCNCPoint3[3195] = {X 0.1542, Y 23.1599, Z -3.8333, A 0.000, B 0.000, C 0.000 }
gfCNCPoint3[3196] = {X -0.3491, Y 22.5478, Z -3.8333, A 0.000, B 0.000, C 0.000 }
gfCNCPoint3[3197] = {X -0.7246, Y 21.8500, Z -3.8333, A 0.000, B 0.000, C 0.000 }
gfCNCPoint3[3198] = {X -3.3966, Y 15.3006, Z -3.8333, A 0.000, B 0.000, C 0.000 }
gfCNCPoint3[3199] = {X -3.6235, Y 14.3620, Z -3.8333, A 0.000, B 0.000, C 0.000 }
gfCNCPoint3[3200] = {X -3.6235, Y 13.3963, Z -3.8333, A 0.000, B 0.000, C 0.000 }
gfCNCPoint3[3201] = {X -3.3966, Y 12.4577, Z -3.8333, A 0.000, B 0.000, C 0.000 }
gfCNCPoint3[3202] = {X -2.9669, Y 11.6159, Z -3.8333, A 0.000, B 0.000, C 0.000 }
gfCNCPoint3[3203] = {X -2.3551, Y 10.8955, Z -3.8333, A 0.000, B 0.000, C 0.000 }
gfCNCPoint3[3204] = {X -1.5940, Y 10.3353, Z -3.8333, A 0.000, B 0.000, C 0.000 }
gfCNCPoint3[3205] = {X -0.9968, Y 9.9945, Z -3.8333, A 0.000, B 0.000, C 0.000 }
gfCNCPoint3[3206] = {X -0.1339, Y 9.6265, Z -3.8333, A 0.000, B 0.000, C 0.000 }
gfCNCPoint3[3207] = {X 0.7902, Y 9.4652, Z -3.8333, A 0.000, B 0.000, C 0.000 }
gfCNCPoint3[3208] = {X 1.7267, Y 9.5193, Z -3.8333, A 0.000, B 0.000, C 0.000 }
gfCNCPoint3[3209] = {X 2.6262, Y 9.7858, Z -3.8333, A 0.000, B 0.000, C 0.000 }
gfCNCPoint3[3210] = {X 3.4400, Y 9.3952, Z -3.8333, A 0.000, B 0.000, C 0.000 }
gfCNCPoint3[3211] = {X 4.2815, Y 9.0685, Z -3.8333, A 0.000, B 0.000, C 0.000 }
gfCNCPoint3[3212] = {X 6.1735, Y 8.4059, Z -3.8333, A 0.000, B 0.000, C 0.000 }
gfCNCPoint3[3213] = {X 8.1157, Y 7.9091, Z -3.8333, A 0.000, B 0.000, C 0.000 }
gfCNCPoint3[3214] = {X 10.0936, Y 7.5816, Z -3.8333, A 0.000, B 0.000, C 0.000 }
gfCNCPoint3[3215] = {X 12.0922, Y 7.4260, Z -3.8333, A 0.000, B 0.000, C 0.000 }
gfCNCPoint3[3216] = {X 14.0969, Y 7.4434, Z -3.8333, A 0.000, B 0.000, C 0.000 }
gfCNCPoint3[3217] = {X 16.0926, Y 7.6337, Z -3.8333, A 0.000, B 0.000, C 0.000 }
gfCNCPoint3[3218] = {X 17.8910, Y 7.9626, Z -3.8333, A 0.000, B 0.000, C 0.000 }
gfCNCPoint3[3219] = {X 19.6443, Y 8.4804, Z -3.8333, A 0.000, B 0.000, C 0.000 }
gfCNCPoint3[3220] = {X 21.3329, Y 9.1812, Z -3.8333, A 0.000, B 0.000, C 0.000 }
gfCNCPoint3[3221] = {X 22.9376, Y 10.0572, Z -3.8333, A 0.000, B 0.000, C 0.000 }
gfCNCPoint3[3222] = {X 24.4404, Y 11.0984, Z -3.8333, A 0.000, B 0.000, C 0.000 }
gfCNCPoint3[3223] = {X 25.5053, Y 12.0295, Z -3.8333, A 0.000, B 0.000, C 0.000 }
gfCNCPoint3[3224] = {X 26.4605, Y 13.0728, Z -3.8333, A 0.000, B 0.000, C 0.000 }
gfCNCPoint3[3225] = {X 27.2944, Y 14.2155, Z -3.8333, A 0.000, B 0.000, C 0.000 }
gfCNCPoint3[3226] = {X 27.9966, Y 15.4435, Z -3.8333, A 0.000, B 0.000, C 0.000 }
gfCNCPoint3[3227] = {X 28.5584, Y 16.7417, Z -3.8333, A 0.000, B 0.000, C 0.000 }
gfCNCPoint3[3228] = {X 29.0249, Y 18.3712, Z -3.8333, A 0.000, B 0.000, C 0.000 }
gfCNCPoint3[3229] = {X 29.3016, Y 20.0434, Z -3.8333, A 0.000, B 0.000, C 0.000 }
gfCNCPoint3[3230] = {X 29.3850, Y 21.7364, Z -3.8333, A 0.000, B 0.000, C 0.000 }
gfCNCPoint3[3231] = {X 29.2740, Y 23.4277, Z -3.8333, A 0.000, B 0.000, C 0.000 }
gfCNCPoint3[3232] = {X 28.9699, Y 25.0952, Z -3.8333, A 0.000, B 0.000, C 0.000 }
gfCNCPoint3[3233] = {X 28.5023, Y 26.6020, Z -3.8333, A 0.000, B 0.000, C 0.000 }
gfCNCPoint3[3234] = {X 27.8320, Y 28.0303, Z -3.8333, A 0.000, B 0.000, C 0.000 }
gfCNCPoint3[3235] = {X 26.9717, Y 29.3528, Z -3.8333, A 0.000, B 0.000, C 0.000 }
gfCNCPoint3[3236] = {X 25.9377, Y 30.5446, Z -3.8333, A 0.000, B 0.000, C 0.000 }
gfCNCPoint3[3237] = {X 24.7498, Y 31.5828, Z -3.8333, A 0.000, B 0.000, C 0.000 }
gfCNCPoint3[3238] = {X 25.0468, Y 31.6499, Z -3.8333, A 0.000, B 0.000, C 0.000 }
gfCNCPoint3[3239] = {X 25.3379, Y 31.7389, Z -3.8333, A 0.000, B 0.000, C 0.000 }
gfCNCPoint3[3240] = {X 26.0572, Y 32.0698, Z -3.8333, A 0.000, B 0.000, C 0.000 }
gfCNCPoint3[3241] = {X 26.6990, Y 32.5334, Z -3.8333, A 0.000, B 0.000, C 0.000 }
gfCNCPoint3[3242] = {X 27.2392, Y 33.1123, Z -3.8333, A 0.000, B 0.000, C 0.000 }
gfCNCPoint3[3243] = {X 27.6575, Y 33.7845, Z -3.8333, A 0.000, B 0.000, C 0.000 }
gfCNCPoint3[3244] = {X 30.6940, Y 40.0576, Z -3.8333, A 0.000, B 0.000, C 0.000 }
gfCNCPoint3[3245] = {X 30.9967, Y 40.9162, Z -3.8333, A 0.000, B 0.000, C 0.000 }
gfCNCPoint3[3246] = {X 31.1015, Y 41.8206, Z -3.8333, A 0.000, B 0.000, C 0.000 }
gfCNCPoint3[3247] = {X 31.0032, Y 42.7257, Z -3.8333, A 0.000, B 0.000, C 0.000 }
gfCNCPoint3[3248] = {X 30.7066, Y 43.5864, Z -3.8333, A 0.000, B 0.000, C 0.000 }
gfCNCPoint3[3249] = {X 30.2265, Y 44.3600, Z -3.8333, A 0.000, B 0.000, C 0.000 }
gfCNCPoint3[3250] = {X 29.5868, Y 45.0078, Z -3.8333, A 0.000, B 0.000, C 0.000 }
gfCNCPoint3[3251] = {X 29.0507, Y 45.4413, Z -3.8333, A 0.000, B 0.000, C 0.000 }
gfCNCPoint3[3252] = {X 28.3671, Y 45.8885, Z -3.8333, A 0.000, B 0.000, C 0.000 }
gfCNCPoint3[3253] = {X 27.6083, Y 46.1911, Z -3.8333, A 0.000, B 0.000, C 0.000 }
gfCNCPoint3[3254] = {X 26.8045, Y 46.3370, Z -3.8333, A 0.000, B 0.000, C 0.000 }
gfCNCPoint3[3255] = {X 25.9877, Y 46.3205, Z -3.8333, A 0.000, B 0.000, C 0.000 }
gfCNCPoint3[3256] = {X 25.1905, Y 46.1422, Z -3.8333, A 0.000, B 0.000, C 0.000 }
gfCNCPoint3[3257] = {X 23.3777, Y 47.1076, Z -3.8333, A 0.000, B 0.000, C 0.000 }
gfCNCPoint3[3258] = {X 21.5007, Y 47.9412, Z -3.8333, A 0.000, B 0.000, C 0.000 }
gfCNCPoint3[3259] = {X 19.5690, Y 48.6388, Z -3.8333, A 0.000, B 0.000, C 0.000 }
gfCNCPoint3[3260] = {X 17.3987, Y 49.2367, Z -3.8333, A 0.000, B 0.000, C 0.000 }
gfCNCPoint3[3261] = {X 15.1797, Y 49.6158, Z -3.8333, A 0.000, B 0.000, C 0.000 }
gfCNCPoint3[3262] = {X 12.9340, Y 49.7724, Z -3.8333, A 0.000, B 0.000, C 0.000 }
gfCNCPoint3[3263] = {X 10.6839, Y 49.7049, Z -3.8333, A 0.000, B 0.000, C 0.000 }
gfCNCPoint3[3264] = {X 8.4516, Y 49.4140, Z -3.8333, A 0.000, B 0.000, C 0.000 }
gfCNCPoint3[3265] = {X 6.5989, Y 48.9851, Z -3.8333, A 0.000, B 0.000, C 0.000 }
gfCNCPoint3[3266] = {X 4.8062, Y 48.3503, Z -3.8333, A 0.000, B 0.000, C 0.000 }
gfCNCPoint3[3267] = {X 3.0965, Y 47.5174, Z -3.8333, A 0.000, B 0.000, C 0.000 }
gfCNCPoint3[3268] = {X 1.4915, Y 46.4973, Z -3.8333, A 0.000, B 0.000, C 0.000 }
gfCNCPoint3[3269] = {X 0.7974, Y 45.9583, Z -3.8333, A 0.000, B 0.000, C 0.000 }
gfCNCPoint3[3270] = {X -0.3147, Y 44.9591, Z -3.8333, A 0.000, B 0.000, C 0.000 }
gfCNCPoint3[3271] = {X -1.3023, Y 43.8366, Z -3.8333, A 0.000, B 0.000, C 0.000 }
gfCNCPoint3[3272] = {X -2.1518, Y 42.6064, Z -3.8333, A 0.000, B 0.000, C 0.000 }
gfCNCPoint3[3273] = {X -2.8515, Y 41.2852, Z -3.8333, A 0.000, B 0.000, C 0.000 }
gfCNCPoint3[3274] = {X -3.3919, Y 39.8912, Z -3.8333, A 0.000, B 0.000, C 0.000 }
gfCNCPoint3[3275] = {X -3.5570, Y 39.3350, Z -3.8333, A 0.000, B 0.000, C 0.000 }
gfCNCPoint3[3276] = {X -3.6965, Y 38.7718, Z -3.8333, A 0.000, B 0.000, C 0.000 }
gfCNCPoint3[3277] = {X -4.5704, Y 34.8685, Z -3.8333, A 0.000, B 0.000, C 0.000 }
gfCNCPoint3[3278] = {X -7.9964, Y 34.7604, Z -3.8333, A 0.000, B 0.000, C 0.000 }
gfCNCPoint3[3279] = {X -7.9964, Y 34.7604, Z -0.8333, A 0.000, B 0.000, C 0.000 }
gfCNCPoint3[3280] = {X -7.9964, Y 34.7604, Z 11.0000, A 0.000, B 0.000, C 0.000 }
gfCNCPoint3[3281] = {X -7.9696, Y 36.4968, Z 11.0000, A 0.000, B 0.000, C 0.000 }
gfCNCPoint3[3282] = {X -7.9696, Y 36.4968, Z -0.8333, A 0.000, B 0.000, C 0.000 }
gfCNCPoint3[3283] = {X -7.9696, Y 36.4968, Z -3.8333, A 0.000, B 0.000, C 0.000 }
gfCNCPoint3[3284] = {X -4.5180, Y 36.2812, Z -3.8333, A 0.000, B 0.000, C 0.000 }
gfCNCPoint3[3285] = {X -3.6965, Y 32.3665, Z -3.8333, A 0.000, B 0.000, C 0.000 }
gfCNCPoint3[3286] = {X -3.5246, Y 31.6406, Z -3.8333, A 0.000, B 0.000, C 0.000 }
gfCNCPoint3[3287] = {X -3.3156, Y 30.9245, Z -3.8333, A 0.000, B 0.000, C 0.000 }
gfCNCPoint3[3288] = {X -3.1439, Y 30.4203, Z -3.8333, A 0.000, B 0.000, C 0.000 }
gfCNCPoint3[3289] = {X -2.9539, Y 29.9228, Z -3.8333, A 0.000, B 0.000, C 0.000 }
gfCNCPoint3[3290] = {X -2.3880, Y 28.7127, Z -3.8333, A 0.000, B 0.000, C 0.000 }
gfCNCPoint3[3291] = {X -1.6730, Y 27.5842, Z -3.8333, A 0.000, B 0.000, C 0.000 }
gfCNCPoint3[3292] = {X -0.8207, Y 26.5556, Z -3.8333, A 0.000, B 0.000, C 0.000 }
gfCNCPoint3[3293] = {X 0.1553, Y 25.6434, Z -3.8333, A 0.000, B 0.000, C 0.000 }
gfCNCPoint3[3294] = {X 1.2392, Y 24.8625, Z -3.8333, A 0.000, B 0.000, C 0.000 }
gfCNCPoint3[3295] = {X 2.4134, Y 24.2255, Z -3.8333, A 0.000, B 0.000, C 0.000 }
gfCNCPoint3[3296] = {X 1.9465, Y 24.1226, Z -3.8333, A 0.000, B 0.000, C 0.000 }
gfCNCPoint3[3297] = {X 1.4951, Y 23.9648, Z -3.8333, A 0.000, B 0.000, C 0.000 }
gfCNCPoint3[3298] = {X 0.8036, Y 23.5918, Z -3.8333, A 0.000, B 0.000, C 0.000 }
gfCNCPoint3[3299] = {X 0.1984, Y 23.0909, Z -3.8333, A 0.000, B 0.000, C 0.000 }
gfCNCPoint3[3300] = {X -0.2973, Y 22.4813, Z -3.8333, A 0.000, B 0.000, C 0.000 }
gfCNCPoint3[3301] = {X -0.6642, Y 21.7866, Z -3.8333, A 0.000, B 0.000, C 0.000 }
gfCNCPoint3[3302] = {X -3.2754, Y 15.3911, Z -3.8333, A 0.000, B 0.000, C 0.000 }
gfCNCPoint3[3303] = {X -3.2990, Y 15.3321, Z -3.8333, A 0.000, B 0.000, C 0.000 }
gfCNCPoint3[3304] = {X -3.3216, Y 15.2727, Z -3.8333, A 0.000, B 0.000, C 0.000 }
gfCNCPoint3[3305] = {X -3.5441, Y 14.3525, Z -3.8333, A 0.000, B 0.000, C 0.000 }
gfCNCPoint3[3306] = {X -3.5441, Y 13.4058, Z -3.8333, A 0.000, B 0.000, C 0.000 }
gfCNCPoint3[3307] = {X -3.3216, Y 12.4855, Z -3.8333, A 0.000, B 0.000, C 0.000 }
gfCNCPoint3[3308] = {X -2.9004, Y 11.6603, Z -3.8333, A 0.000, B 0.000, C 0.000 }
gfCNCPoint3[3309] = {X -2.3006, Y 10.9540, Z -3.8333, A 0.000, B 0.000, C 0.000 }
gfCNCPoint3[3310] = {X -1.5544, Y 10.4048, Z -3.8333, A 0.000, B 0.000, C 0.000 }
gfCNCPoint3[3311] = {X -0.9063, Y 10.0355, Z -3.8333, A 0.000, B 0.000, C 0.000 }
gfCNCPoint3[3312] = {X -0.0600, Y 9.6884, Z -3.8333, A 0.000, B 0.000, C 0.000 }
gfCNCPoint3[3313] = {X 0.8429, Y 9.5426, Z -3.8333, A 0.000, B 0.000, C 0.000 }
gfCNCPoint3[3314] = {X 1.7554, Y 9.6057, Z -3.8333, A 0.000, B 0.000, C 0.000 }
gfCNCPoint3[3315] = {X 2.6297, Y 9.8745, Z -3.8333, A 0.000, B 0.000, C 0.000 }
gfCNCPoint3[3316] = {X 2.7107, Y 9.8318, Z -3.8333, A 0.000, B 0.000, C 0.000 }
gfCNCPoint3[3317] = {X 2.7920, Y 9.7897, Z -3.8333, A 0.000, B 0.000, C 0.000 }
gfCNCPoint3[3318] = {X 3.5435, Y 9.4376, Z -3.8333, A 0.000, B 0.000, C 0.000 }
gfCNCPoint3[3319] = {X 4.3182, Y 9.1400, Z -3.8333, A 0.000, B 0.000, C 0.000 }
gfCNCPoint3[3320] = {X 6.2027, Y 8.4807, Z -3.8333, A 0.000, B 0.000, C 0.000 }
gfCNCPoint3[3321] = {X 8.1371, Y 7.9863, Z -3.8333, A 0.000, B 0.000, C 0.000 }
gfCNCPoint3[3322] = {X 10.1070, Y 7.6606, Z -3.8333, A 0.000, B 0.000, C 0.000 }
gfCNCPoint3[3323] = {X 12.0975, Y 7.5059, Z -3.8333, A 0.000, B 0.000, C 0.000 }
gfCNCPoint3[3324] = {X 14.0940, Y 7.5234, Z -3.8333, A 0.000, B 0.000, C 0.000 }
gfCNCPoint3[3325] = {X 16.0816, Y 7.7129, Z -3.8333, A 0.000, B 0.000, C 0.000 }
gfCNCPoint3[3326] = {X 16.4815, Y 7.7686, Z -3.8333, A 0.000, B 0.000, C 0.000 }
gfCNCPoint3[3327] = {X 18.1854, Y 8.1178, Z -3.8333, A 0.000, B 0.000, C 0.000 }
gfCNCPoint3[3328] = {X 19.8450, Y 8.6378, Z -3.8333, A 0.000, B 0.000, C 0.000 }
gfCNCPoint3[3329] = {X 21.4435, Y 9.3235, Z -3.8333, A 0.000, B 0.000, C 0.000 }
gfCNCPoint3[3330] = {X 22.9641, Y 10.1677, Z -3.8333, A 0.000, B 0.000, C 0.000 }
gfCNCPoint3[3331] = {X 24.3914, Y 11.1616, Z -3.8333, A 0.000, B 0.000, C 0.000 }
gfCNCPoint3[3332] = {X 25.4494, Y 12.0868, Z -3.8333, A 0.000, B 0.000, C 0.000 }
gfCNCPoint3[3333] = {X 26.3986, Y 13.1235, Z -3.8333, A 0.000, B 0.000, C 0.000 }
gfCNCPoint3[3334] = {X 27.2271, Y 14.2588, Z -3.8333, A 0.000, B 0.000, C 0.000 }
gfCNCPoint3[3335] = {X 27.9248, Y 15.4789, Z -3.8333, A 0.000, B 0.000, C 0.000 }
gfCNCPoint3[3336] = {X 28.4831, Y 16.7687, Z -3.8333, A 0.000, B 0.000, C 0.000 }
gfCNCPoint3[3337] = {X 28.9470, Y 18.3896, Z -3.8333, A 0.000, B 0.000, C 0.000 }
gfCNCPoint3[3338] = {X 29.2222, Y 20.0529, Z -3.8333, A 0.000, B 0.000, C 0.000 }
gfCNCPoint3[3339] = {X 29.3050, Y 21.7368, Z -3.8333, A 0.000, B 0.000, C 0.000 }
gfCNCPoint3[3340] = {X 29.1944, Y 23.4191, Z -3.8333, A 0.000, B 0.000, C 0.000 }
gfCNCPoint3[3341] = {X 28.8919, Y 25.0777, Z -3.8333, A 0.000, B 0.000, C 0.000 }
gfCNCPoint3[3342] = {X 28.4138, Y 26.6088, Z -3.8333, A 0.000, B 0.000, C 0.000 }
gfCNCPoint3[3343] = {X 27.7251, Y 28.0574, Z -3.8333, A 0.000, B 0.000, C 0.000 }
gfCNCPoint3[3344] = {X 26.8393, Y 29.3947, Z -3.8333, A 0.000, B 0.000, C 0.000 }
gfCNCPoint3[3345] = {X 25.7741, Y 30.5940, Z -3.8333, A 0.000, B 0.000, C 0.000 }
gfCNCPoint3[3346] = {X 24.5508, Y 31.6315, Z -3.8333, A 0.000, B 0.000, C 0.000 }
gfCNCPoint3[3347] = {X 24.9357, Y 31.7043, Z -3.8333, A 0.000, B 0.000, C 0.000 }
gfCNCPoint3[3348] = {X 25.3117, Y 31.8145, Z -3.8333, A 0.000, B 0.000, C 0.000 }
gfCNCPoint3[3349] = {X 26.0243, Y 32.1432, Z -3.8333, A 0.000, B 0.000, C 0.000 }
gfCNCPoint3[3350] = {X 26.6590, Y 32.6048, Z -3.8333, A 0.000, B 0.000, C 0.000 }
gfCNCPoint3[3351] = {X 27.1913, Y 33.1814, Z -3.8333, A 0.000, B 0.000, C 0.000 }
gfCNCPoint3[3352] = {X 27.6008, Y 33.8508, Z -3.8333, A 0.000, B 0.000, C 0.000 }
gfCNCPoint3[3353] = {X 30.6220, Y 40.0925, Z -3.8333, A 0.000, B 0.000, C 0.000 }
gfCNCPoint3[3354] = {X 30.9188, Y 40.9342, Z -3.8333, A 0.000, B 0.000, C 0.000 }
gfCNCPoint3[3355] = {X 31.0215, Y 41.8209, Z -3.8333, A 0.000, B 0.000, C 0.000 }
gfCNCPoint3[3356] = {X 30.9251, Y 42.7082, Z -3.8333, A 0.000, B 0.000, C 0.000 }
gfCNCPoint3[3357] = {X 30.6343, Y 43.5521, Z -3.8333, A 0.000, B 0.000, C 0.000 }
gfCNCPoint3[3358] = {X 30.1637, Y 44.3105, Z -3.8333, A 0.000, B 0.000, C 0.000 }
gfCNCPoint3[3359] = {X 29.5365, Y 44.9456, Z -3.8333, A 0.000, B 0.000, C 0.000 }
gfCNCPoint3[3360] = {X 29.0005, Y 45.3790, Z -3.8333, A 0.000, B 0.000, C 0.000 }
gfCNCPoint3[3361] = {X 28.3238, Y 45.8208, Z -3.8333, A 0.000, B 0.000, C 0.000 }
gfCNCPoint3[3362] = {X 27.5724, Y 46.1181, Z -3.8333, A 0.000, B 0.000, C 0.000 }
gfCNCPoint3[3363] = {X 26.7767, Y 46.2589, Z -3.8333, A 0.000, B 0.000, C 0.000 }
gfCNCPoint3[3364] = {X 25.9689, Y 46.2375, Z -3.8333, A 0.000, B 0.000, C 0.000 }
gfCNCPoint3[3365] = {X 25.1817, Y 46.0549, Z -3.8333, A 0.000, B 0.000, C 0.000 }
gfCNCPoint3[3366] = {X 25.1059, Y 46.0987, Z -3.8333, A 0.000, B 0.000, C 0.000 }
gfCNCPoint3[3367] = {X 25.0300, Y 46.1424, Z -3.8333, A 0.000, B 0.000, C 0.000 }
gfCNCPoint3[3368] = {X 23.2583, Y 47.0766, Z -3.8333, A 0.000, B 0.000, C 0.000 }
gfCNCPoint3[3369] = {X 21.4258, Y 47.8850, Z -3.8333, A 0.000, B 0.000, C 0.000 }
gfCNCPoint3[3370] = {X 19.5414, Y 48.5637, Z -3.8333, A 0.000, B 0.000, C 0.000 }
gfCNCPoint3[3371] = {X 19.3877, Y 48.6154, Z -3.8333, A 0.000, B 0.000, C 0.000 }
gfCNCPoint3[3372] = {X 17.2526, Y 49.1882, Z -3.8333, A 0.000, B 0.000, C 0.000 }
gfCNCPoint3[3373] = {X 15.0715, Y 49.5490, Z -3.8333, A 0.000, B 0.000, C 0.000 }
gfCNCPoint3[3374] = {X 12.8656, Y 49.6943, Z -3.8333, A 0.000, B 0.000, C 0.000 }
gfCNCPoint3[3375] = {X 10.6561, Y 49.6227, Z -3.8333, A 0.000, B 0.000, C 0.000 }
gfCNCPoint3[3376] = {X 8.4642, Y 49.3350, Z -3.8333, A 0.000, B 0.000, C 0.000 }
gfCNCPoint3[3377] = {X 6.6209, Y 48.9082, Z -3.8333, A 0.000, B 0.000, C 0.000 }
gfCNCPoint3[3378] = {X 4.8374, Y 48.2766, Z -3.8333, A 0.000, B 0.000, C 0.000 }
gfCNCPoint3[3379] = {X 3.1363, Y 47.4480, Z -3.8333, A 0.000, B 0.000, C 0.000 }
gfCNCPoint3[3380] = {X 1.5394, Y 46.4332, Z -3.8333, A 0.000, B 0.000, C 0.000 }
gfCNCPoint3[3381] = {X 0.8469, Y 45.8954, Z -3.8333, A 0.000, B 0.000, C 0.000 }
gfCNCPoint3[3382] = {X -0.2581, Y 44.9025, Z -3.8333, A 0.000, B 0.000, C 0.000 }
gfCNCPoint3[3383] = {X -1.2394, Y 43.7872, Z -3.8333, A 0.000, B 0.000, C 0.000 }
gfCNCPoint3[3384] = {X -2.0835, Y 42.5647, Z -3.8333, A 0.000, B 0.000, C 0.000 }
gfCNCPoint3[3385] = {X -2.7788, Y 41.2518, Z -3.8333, A 0.000, B 0.000, C 0.000 }
gfCNCPoint3[3386] = {X -3.3158, Y 39.8667, Z -3.8333, A 0.000, B 0.000, C 0.000 }
gfCNCPoint3[3387] = {X -3.5287, Y 39.1287, Z -3.8333, A 0.000, B 0.000, C 0.000 }
gfCNCPoint3[3388] = {X -3.6965, Y 38.3791, Z -3.8333, A 0.000, B 0.000, C 0.000 }
gfCNCPoint3[3389] = {X -4.4520, Y 34.4511, Z -3.8333, A 0.000, B 0.000, C 0.000 }
gfCNCPoint3[3390] = {X -7.9726, Y 34.2408, Z -3.8333, A 0.000, B 0.000, C 0.000 }
gfCNCPoint3[3391] = {X -7.9726, Y 34.2408, Z -0.8333, A 0.000, B 0.000, C 0.000 }
gfCNCPoint3[3392] = {X -7.9726, Y 34.2408, Z 11.0000, A 0.000, B 0.000, C 0.000 }
gfCNCPoint3[3393] = {X 39.8251, Y 26.3830, Z 11.0000, A 0.000, B 0.000, C 0.000 }
gfCNCPoint3[3394] = {X 39.8251, Y 26.3830, Z -0.8333, A 0.000, B 0.000, C 0.000 }
gfCNCPoint3[3395] = {X 39.8251, Y 26.3830, Z -3.8333, A 0.000, B 0.000, C 0.000 }
gfCNCPoint3[3396] = {X 43.6485, Y 27.8070, Z -3.8333, A 0.000, B 0.000, C 0.000 }
gfCNCPoint3[3397] = {X 48.2901, Y 15.3446, Z -3.8333, A 0.000, B 0.000, C 0.000 }
gfCNCPoint3[3398] = {X 47.9079, Y 14.6186, Z -3.8333, A 0.000, B 0.000, C 0.000 }
gfCNCPoint3[3399] = {X 47.6698, Y 13.8334, Z -3.8333, A 0.000, B 0.000, C 0.000 }
gfCNCPoint3[3400] = {X 47.5844, Y 13.0173, Z -3.8333, A 0.000, B 0.000, C 0.000 }
gfCNCPoint3[3401] = {X 47.5842, Y 12.1868, Z -3.8333, A 0.000, B 0.000, C 0.000 }
gfCNCPoint3[3402] = {X 47.6925, Y 11.2255, Z -3.8333, A 0.000, B 0.000, C 0.000 }
gfCNCPoint3[3403] = {X 48.0120, Y 10.3125, Z -3.8333, A 0.000, B 0.000, C 0.000 }
gfCNCPoint3[3404] = {X 48.5267, Y 9.4933, Z -3.8333, A 0.000, B 0.000, C 0.000 }
gfCNCPoint3[3405] = {X 49.2107, Y 8.8093, Z -3.8333, A 0.000, B 0.000, C 0.000 }
gfCNCPoint3[3406] = {X 50.0298, Y 8.2946, Z -3.8333, A 0.000, B 0.000, C 0.000 }
gfCNCPoint3[3407] = {X 50.9429, Y 7.9751, Z -3.8333, A 0.000, B 0.000, C 0.000 }
gfCNCPoint3[3408] = {X 51.9042, Y 7.8668, Z -3.8333, A 0.000, B 0.000, C 0.000 }
gfCNCPoint3[3409] = {X 59.6221, Y 7.8668, Z -3.8333, A 0.000, B 0.000, C 0.000 }
gfCNCPoint3[3410] = {X 60.5834, Y 7.9751, Z -3.8333, A 0.000, B 0.000, C 0.000 }
gfCNCPoint3[3411] = {X 61.4965, Y 8.2946, Z -3.8333, A 0.000, B 0.000, C 0.000 }
gfCNCPoint3[3412] = {X 62.3156, Y 8.8093, Z -3.8333, A 0.000, B 0.000, C 0.000 }
gfCNCPoint3[3413] = {X 62.9996, Y 9.4933, Z -3.8333, A 0.000, B 0.000, C 0.000 }
gfCNCPoint3[3414] = {X 63.5143, Y 10.3124, Z -3.8333, A 0.000, B 0.000, C 0.000 }
gfCNCPoint3[3415] = {X 63.8338, Y 11.2255, Z -3.8333, A 0.000, B 0.000, C 0.000 }
gfCNCPoint3[3416] = {X 63.9421, Y 12.1868, Z -3.8333, A 0.000, B 0.000, C 0.000 }
gfCNCPoint3[3417] = {X 63.9421, Y 12.9781, Z -3.8333, A 0.000, B 0.000, C 0.000 }
gfCNCPoint3[3418] = {X 63.8583, Y 13.8248, Z -3.8333, A 0.000, B 0.000, C 0.000 }
gfCNCPoint3[3419] = {X 63.6102, Y 14.6386, Z -3.8333, A 0.000, B 0.000, C 0.000 }
gfCNCPoint3[3420] = {X 63.2074, Y 15.3880, Z -3.8333, A 0.000, B 0.000, C 0.000 }
gfCNCPoint3[3421] = {X 63.4255, Y 15.9633, Z -3.8333, A 0.000, B 0.000, C 0.000 }
gfCNCPoint3[3422] = {X 66.2401, Y 23.4314, Z -3.8333, A 0.000, B 0.000, C 0.000 }
gfCNCPoint3[3423] = {X 72.2094, Y 39.5004, Z -3.8333, A 0.000, B 0.000, C 0.000 }
gfCNCPoint3[3424] = {X 72.5146, Y 40.2681, Z -3.8333, A 0.000, B 0.000, C 0.000 }
gfCNCPoint3[3425] = {X 73.3591, Y 40.7699, Z -3.8333, A 0.000, B 0.000, C 0.000 }
gfCNCPoint3[3426] = {X 74.0684, Y 41.4495, Z -3.8333, A 0.000, B 0.000, C 0.000 }
gfCNCPoint3[3427] = {X 74.6059, Y 42.2718, Z -3.8333, A 0.000, B 0.000, C 0.000 }
gfCNCPoint3[3428] = {X 74.9436, Y 43.1942, Z -3.8333, A 0.000, B 0.000, C 0.000 }
gfCNCPoint3[3429] = {X 75.0643, Y 44.1692, Z -3.8333, A 0.000, B 0.000, C 0.000 }
gfCNCPoint3[3430] = {X 75.0645, Y 45.0000, Z -3.8333, A 0.000, B 0.000, C 0.000 }
gfCNCPoint3[3431] = {X 74.9561, Y 45.9613, Z -3.8333, A 0.000, B 0.000, C 0.000 }
gfCNCPoint3[3432] = {X 74.6366, Y 46.8744, Z -3.8333, A 0.000, B 0.000, C 0.000 }
gfCNCPoint3[3433] = {X 74.1220, Y 47.6935, Z -3.8333, A 0.000, B 0.000, C 0.000 }
gfCNCPoint3[3434] = {X 73.4379, Y 48.3775, Z -3.8333, A 0.000, B 0.000, C 0.000 }
gfCNCPoint3[3435] = {X 72.6188, Y 48.8922, Z -3.8333, A 0.000, B 0.000, C 0.000 }
gfCNCPoint3[3436] = {X 71.7057, Y 49.2117, Z -3.8333, A 0.000, B 0.000, C 0.000 }
gfCNCPoint3[3437] = {X 70.7445, Y 49.3200, Z -3.8333, A 0.000, B 0.000, C 0.000 }
gfCNCPoint3[3438] = {X 64.1851, Y 49.3200, Z -3.8333, A 0.000, B 0.000, C 0.000 }
gfCNCPoint3[3439] = {X 63.2238, Y 49.2117, Z -3.8333, A 0.000, B 0.000, C 0.000 }
gfCNCPoint3[3440] = {X 62.3108, Y 48.8922, Z -3.8333, A 0.000, B 0.000, C 0.000 }
gfCNCPoint3[3441] = {X 61.4917, Y 48.3775, Z -3.8333, A 0.000, B 0.000, C 0.000 }
gfCNCPoint3[3442] = {X 60.8076, Y 47.6935, Z -3.8333, A 0.000, B 0.000, C 0.000 }
gfCNCPoint3[3443] = {X 60.2929, Y 46.8744, Z -3.8333, A 0.000, B 0.000, C 0.000 }
gfCNCPoint3[3444] = {X 59.9734, Y 45.9613, Z -3.8333, A 0.000, B 0.000, C 0.000 }
gfCNCPoint3[3445] = {X 59.8651, Y 45.0000, Z -3.8333, A 0.000, B 0.000, C 0.000 }
gfCNCPoint3[3446] = {X 59.8651, Y 44.2085, Z -3.8333, A 0.000, B 0.000, C 0.000 }
gfCNCPoint3[3447] = {X 59.9519, Y 43.3501, Z -3.8333, A 0.000, B 0.000, C 0.000 }
gfCNCPoint3[3448] = {X 60.2076, Y 42.5260, Z -3.8333, A 0.000, B 0.000, C 0.000 }
gfCNCPoint3[3449] = {X 60.6219, Y 41.7692, Z -3.8333, A 0.000, B 0.000, C 0.000 }
gfCNCPoint3[3450] = {X 60.0071, Y 40.0892, Z -3.8333, A 0.000, B 0.000, C 0.000 }
gfCNCPoint3[3451] = {X 52.0770, Y 40.0892, Z -3.8333, A 0.000, B 0.000, C 0.000 }
gfCNCPoint3[3452] = {X 51.3343, Y 42.0845, Z -3.8333, A 0.000, B 0.000, C 0.000 }
gfCNCPoint3[3453] = {X 51.3375, Y 42.0897, Z -3.8333, A 0.000, B 0.000, C 0.000 }
gfCNCPoint3[3454] = {X 51.6389, Y 42.7492, Z -3.8333, A 0.000, B 0.000, C 0.000 }
gfCNCPoint3[3455] = {X 51.8257, Y 43.4499, Z -3.8333, A 0.000, B 0.000, C 0.000 }
gfCNCPoint3[3456] = {X 51.8928, Y 44.1720, Z -3.8333, A 0.000, B 0.000, C 0.000 }
gfCNCPoint3[3457] = {X 51.8929, Y 45.0000, Z -3.8333, A 0.000, B 0.000, C 0.000 }
gfCNCPoint3[3458] = {X 51.7846, Y 45.9613, Z -3.8333, A 0.000, B 0.000, C 0.000 }
gfCNCPoint3[3459] = {X 51.4651, Y 46.8744, Z -3.8333, A 0.000, B 0.000, C 0.000 }
gfCNCPoint3[3460] = {X 50.9504, Y 47.6935, Z -3.8333, A 0.000, B 0.000, C 0.000 }
gfCNCPoint3[3461] = {X 50.2664, Y 48.3775, Z -3.8333, A 0.000, B 0.000, C 0.000 }
gfCNCPoint3[3462] = {X 49.4473, Y 48.8922, Z -3.8333, A 0.000, B 0.000, C 0.000 }
gfCNCPoint3[3463] = {X 48.5342, Y 49.2117, Z -3.8333, A 0.000, B 0.000, C 0.000 }
gfCNCPoint3[3464] = {X 47.5729, Y 49.3200, Z -3.8333, A 0.000, B 0.000, C 0.000 }
gfCNCPoint3[3465] = {X 40.6393, Y 49.3200, Z -3.8333, A 0.000, B 0.000, C 0.000 }
gfCNCPoint3[3466] = {X 39.6780, Y 49.2117, Z -3.8333, A 0.000, B 0.000, C 0.000 }
gfCNCPoint3[3467] = {X 38.7649, Y 48.8922, Z -3.8333, A 0.000, B 0.000, C 0.000 }
gfCNCPoint3[3468] = {X 37.9458, Y 48.3775, Z -3.8333, A 0.000, B 0.000, C 0.000 }
gfCNCPoint3[3469] = {X 37.2618, Y 47.6935, Z -3.8333, A 0.000, B 0.000, C 0.000 }
gfCNCPoint3[3470] = {X 36.7471, Y 46.8744, Z -3.8333, A 0.000, B 0.000, C 0.000 }
gfCNCPoint3[3471] = {X 36.4276, Y 45.9613, Z -3.8333, A 0.000, B 0.000, C 0.000 }
gfCNCPoint3[3472] = {X 36.3193, Y 45.0000, Z -3.8333, A 0.000, B 0.000, C 0.000 }
gfCNCPoint3[3473] = {X 36.3193, Y 44.2086, Z -3.8333, A 0.000, B 0.000, C 0.000 }
gfCNCPoint3[3474] = {X 36.4360, Y 43.2114, Z -3.8333, A 0.000, B 0.000, C 0.000 }
gfCNCPoint3[3475] = {X 36.7798, Y 42.2680, Z -3.8333, A 0.000, B 0.000, C 0.000 }
gfCNCPoint3[3476] = {X 37.3320, Y 41.4295, Z -3.8333, A 0.000, B 0.000, C 0.000 }
gfCNCPoint3[3477] = {X 38.0630, Y 40.7411, Z -3.8333, A 0.000, B 0.000, C 0.000 }
gfCNCPoint3[3478] = {X 38.9330, Y 40.2400, Z -3.8333, A 0.000, B 0.000, C 0.000 }
gfCNCPoint3[3479] = {X 39.5237, Y 38.8447, Z -3.8333, A 0.000, B 0.000, C 0.000 }
gfCNCPoint3[3480] = {X 40.0647, Y 37.4293, Z -3.8333, A 0.000, B 0.000, C 0.000 }
gfCNCPoint3[3481] = {X 43.6485, Y 27.8070, Z -3.8333, A 0.000, B 0.000, C 0.000 }
gfCNCPoint3[3482] = {X 39.9001, Y 26.4109, Z -3.8333, A 0.000, B 0.000, C 0.000 }
gfCNCPoint3[3483] = {X 43.7235, Y 27.8349, Z -3.8333, A 0.000, B 0.000, C 0.000 }
gfCNCPoint3[3484] = {X 48.3793, Y 15.3344, Z -3.8333, A 0.000, B 0.000, C 0.000 }
gfCNCPoint3[3485] = {X 47.9922, Y 14.6130, Z -3.8333, A 0.000, B 0.000, C 0.000 }
gfCNCPoint3[3486] = {X 47.7508, Y 13.8307, Z -3.8333, A 0.000, B 0.000, C 0.000 }
gfCNCPoint3[3487] = {X 47.6644, Y 13.0166, Z -3.8333, A 0.000, B 0.000, C 0.000 }
gfCNCPoint3[3488] = {X 47.6642, Y 12.1868, Z -3.8333, A 0.000, B 0.000, C 0.000 }
gfCNCPoint3[3489] = {X 47.7705, Y 11.2433, Z -3.8333, A 0.000, B 0.000, C 0.000 }
gfCNCPoint3[3490] = {X 48.0841, Y 10.3472, Z -3.8333, A 0.000, B 0.000, C 0.000 }
gfCNCPoint3[3491] = {X 48.5893, Y 9.5432, Z -3.8333, A 0.000, B 0.000, C 0.000 }
gfCNCPoint3[3492] = {X 49.2606, Y 8.8719, Z -3.8333, A 0.000, B 0.000, C 0.000 }
gfCNCPoint3[3493] = {X 50.0646, Y 8.3667, Z -3.8333, A 0.000, B 0.000, C 0.000 }
gfCNCPoint3[3494] = {X 50.9607, Y 8.0531, Z -3.8333, A 0.000, B 0.000, C 0.000 }
gfCNCPoint3[3495] = {X 51.9042, Y 7.9468, Z -3.8333, A 0.000, B 0.000, C 0.000 }
gfCNCPoint3[3496] = {X 59.6221, Y 7.9468, Z -3.8333, A 0.000, B 0.000, C 0.000 }
gfCNCPoint3[3497] = {X 60.5656, Y 8.0531, Z -3.8333, A 0.000, B 0.000, C 0.000 }
gfCNCPoint3[3498] = {X 61.4618, Y 8.3667, Z -3.8333, A 0.000, B 0.000, C 0.000 }
gfCNCPoint3[3499] = {X 62.2657, Y 8.8718, Z -3.8333, A 0.000, B 0.000, C 0.000 }
gfCNCPoint3[3500] = {X 62.9371, Y 9.5432, Z -3.8333, A 0.000, B 0.000, C 0.000 }
gfCNCPoint3[3501] = {X 63.4422, Y 10.3471, Z -3.8333, A 0.000, B 0.000, C 0.000 }
gfCNCPoint3[3502] = {X 63.7558, Y 11.2433, Z -3.8333, A 0.000, B 0.000, C 0.000 }
gfCNCPoint3[3503] = {X 63.8621, Y 12.1868, Z -3.8333, A 0.000, B 0.000, C 0.000 }
gfCNCPoint3[3504] = {X 63.8621, Y 12.9781, Z -3.8333, A 0.000, B 0.000, C 0.000 }
gfCNCPoint3[3505] = {X 63.7772, Y 13.8226, Z -3.8333, A 0.000, B 0.000, C 0.000 }
gfCNCPoint3[3506] = {X 63.5257, Y 14.6332, Z -3.8333, A 0.000, B 0.000, C 0.000 }
gfCNCPoint3[3507] = {X 63.1179, Y 15.3774, Z -3.8333, A 0.000, B 0.000, C 0.000 }
gfCNCPoint3[3508] = {X 63.3506, Y 15.9916, Z -3.8333, A 0.000, B 0.000, C 0.000 }
gfCNCPoint3[3509] = {X 66.1652, Y 23.4595, Z -3.8333, A 0.000, B 0.000, C 0.000 }
gfCNCPoint3[3510] = {X 72.1347, Y 39.5291, Z -3.8333, A 0.000, B 0.000, C 0.000 }
gfCNCPoint3[3511] = {X 72.4523, Y 40.3279, Z -3.8333, A 0.000, B 0.000, C 0.000 }
gfCNCPoint3[3512] = {X 73.2901, Y 40.8180, Z -3.8333, A 0.000, B 0.000, C 0.000 }
gfCNCPoint3[3513] = {X 73.9944, Y 41.4857, Z -3.8333, A 0.000, B 0.000, C 0.000 }
gfCNCPoint3[3514] = {X 74.5285, Y 42.2961, Z -3.8333, A 0.000, B 0.000, C 0.000 }
gfCNCPoint3[3515] = {X 74.8644, Y 43.2068, Z -3.8333, A 0.000, B 0.000, C 0.000 }
gfCNCPoint3[3516] = {X 74.9843, Y 44.1699, Z -3.8333, A 0.000, B 0.000, C 0.000 }
gfCNCPoint3[3517] = {X 74.9845, Y 45.0000, Z -3.8333, A 0.000, B 0.000, C 0.000 }
gfCNCPoint3[3518] = {X 74.8782, Y 45.9435, Z -3.8333, A 0.000, B 0.000, C 0.000 }
gfCNCPoint3[3519] = {X 74.5646, Y 46.8397, Z -3.8333, A 0.000, B 0.000, C 0.000 }
gfCNCPoint3[3520] = {X 74.0594, Y 47.6436, Z -3.8333, A 0.000, B 0.000, C 0.000 }
gfCNCPoint3[3521] = {X 73.3881, Y 48.3150, Z -3.8333, A 0.000, B 0.000, C 0.000 }
gfCNCPoint3[3522] = {X 72.5841, Y 48.8201, Z -3.8333, A 0.000, B 0.000, C 0.000 }
gfCNCPoint3[3523] = {X 71.6879, Y 49.1337, Z -3.8333, A 0.000, B 0.000, C 0.000 }
gfCNCPoint3[3524] = {X 70.7445, Y 49.2400, Z -3.8333, A 0.000, B 0.000, C 0.000 }
gfCNCPoint3[3525] = {X 64.1851, Y 49.2400, Z -3.8333, A 0.000, B 0.000, C 0.000 }
gfCNCPoint3[3526] = {X 63.2416, Y 49.1337, Z -3.8333, A 0.000, B 0.000, C 0.000 }
gfCNCPoint3[3527] = {X 62.3455, Y 48.8201, Z -3.8333, A 0.000, B 0.000, C 0.000 }
gfCNCPoint3[3528] = {X 61.5415, Y 48.3150, Z -3.8333, A 0.000, B 0.000, C 0.000 }
gfCNCPoint3[3529] = {X 60.8702, Y 47.6436, Z -3.8333, A 0.000, B 0.000, C 0.000 }
gfCNCPoint3[3530] = {X 60.3650, Y 46.8397, Z -3.8333, A 0.000, B 0.000, C 0.000 }
gfCNCPoint3[3531] = {X 60.0514, Y 45.9435, Z -3.8333, A 0.000, B 0.000, C 0.000 }
gfCNCPoint3[3532] = {X 59.9451, Y 45.0000, Z -3.8333, A 0.000, B 0.000, C 0.000 }
gfCNCPoint3[3533] = {X 59.9451, Y 44.2085, Z -3.8333, A 0.000, B 0.000, C 0.000 }
gfCNCPoint3[3534] = {X 60.0331, Y 43.3526, Z -3.8333, A 0.000, B 0.000, C 0.000 }
gfCNCPoint3[3535] = {X 60.2920, Y 42.5320, Z -3.8333, A 0.000, B 0.000, C 0.000 }
gfCNCPoint3[3536] = {X 60.7112, Y 41.7807, Z -3.8333, A 0.000, B 0.000, C 0.000 }
gfCNCPoint3[3537] = {X 60.0630, Y 40.0092, Z -3.8333, A 0.000, B 0.000, C 0.000 }
gfCNCPoint3[3538] = {X 52.0215, Y 40.0092, Z -3.8333, A 0.000, B 0.000, C 0.000 }
gfCNCPoint3[3539] = {X 51.2459, Y 42.0927, Z -3.8333, A 0.000, B 0.000, C 0.000 }
gfCNCPoint3[3540] = {X 51.2683, Y 42.1299, Z -3.8333, A 0.000, B 0.000, C 0.000 }
gfCNCPoint3[3541] = {X 51.5639, Y 42.7770, Z -3.8333, A 0.000, B 0.000, C 0.000 }
gfCNCPoint3[3542] = {X 51.7471, Y 43.4643, Z -3.8333, A 0.000, B 0.000, C 0.000 }
gfCNCPoint3[3543] = {X 51.8128, Y 44.1726, Z -3.8333, A 0.000, B 0.000, C 0.000 }
gfCNCPoint3[3544] = {X 51.8129, Y 45.0000, Z -3.8333, A 0.000, B 0.000, C 0.000 }
gfCNCPoint3[3545] = {X 51.7066, Y 45.9435, Z -3.8333, A 0.000, B 0.000, C 0.000 }
gfCNCPoint3[3546] = {X 51.3930, Y 46.8397, Z -3.8333, A 0.000, B 0.000, C 0.000 }
gfCNCPoint3[3547] = {X 50.8879, Y 47.6436, Z -3.8333, A 0.000, B 0.000, C 0.000 }
gfCNCPoint3[3548] = {X 50.2165, Y 48.3150, Z -3.8333, A 0.000, B 0.000, C 0.000 }
gfCNCPoint3[3549] = {X 49.4126, Y 48.8201, Z -3.8333, A 0.000, B 0.000, C 0.000 }
gfCNCPoint3[3550] = {X 48.5164, Y 49.1337, Z -3.8333, A 0.000, B 0.000, C 0.000 }
gfCNCPoint3[3551] = {X 47.5729, Y 49.2400, Z -3.8333, A 0.000, B 0.000, C 0.000 }
gfCNCPoint3[3552] = {X 40.6393, Y 49.2400, Z -3.8333, A 0.000, B 0.000, C 0.000 }
gfCNCPoint3[3553] = {X 39.6958, Y 49.1337, Z -3.8333, A 0.000, B 0.000, C 0.000 }
gfCNCPoint3[3554] = {X 38.7996, Y 48.8201, Z -3.8333, A 0.000, B 0.000, C 0.000 }
gfCNCPoint3[3555] = {X 37.9957, Y 48.3150, Z -3.8333, A 0.000, B 0.000, C 0.000 }
gfCNCPoint3[3556] = {X 37.3243, Y 47.6436, Z -3.8333, A 0.000, B 0.000, C 0.000 }
gfCNCPoint3[3557] = {X 36.8192, Y 46.8397, Z -3.8333, A 0.000, B 0.000, C 0.000 }
gfCNCPoint3[3558] = {X 36.5056, Y 45.9435, Z -3.8333, A 0.000, B 0.000, C 0.000 }
gfCNCPoint3[3559] = {X 36.3993, Y 45.0000, Z -3.8333, A 0.000, B 0.000, C 0.000 }
gfCNCPoint3[3560] = {X 36.3993, Y 44.2086, Z -3.8333, A 0.000, B 0.000, C 0.000 }
gfCNCPoint3[3561] = {X 36.5153, Y 43.2238, Z -3.8333, A 0.000, B 0.000, C 0.000 }
gfCNCPoint3[3562] = {X 36.8569, Y 42.2928, Z -3.8333, A 0.000, B 0.000, C 0.000 }
gfCNCPoint3[3563] = {X 37.4054, Y 41.4667, Z -3.8333, A 0.000, B 0.000, C 0.000 }
gfCNCPoint3[3564] = {X 38.1307, Y 40.7905, Z -3.8333, A 0.000, B 0.000, C 0.000 }
gfCNCPoint3[3565] = {X 38.9933, Y 40.3013, Z -3.8333, A 0.000, B 0.000, C 0.000 }
gfCNCPoint3[3566] = {X 39.5921, Y 38.8892, Z -3.8333, A 0.000, B 0.000, C 0.000 }
gfCNCPoint3[3567] = {X 40.1399, Y 37.4566, Z -3.8333, A 0.000, B 0.000, C 0.000 }
gfCNCPoint3[3568] = {X 43.7235, Y 27.8349, Z -3.8333, A 0.000, B 0.000, C 0.000 }
gfCNCPoint3[3569] = {X 39.9751, Y 26.4388, Z -3.8333, A 0.000, B 0.000, C 0.000 }
gfCNCPoint3[3570] = {X 43.7985, Y 27.8628, Z -3.8333, A 0.000, B 0.000, C 0.000 }
gfCNCPoint3[3571] = {X 48.4687, Y 15.3238, Z -3.8333, A 0.000, B 0.000, C 0.000 }
gfCNCPoint3[3572] = {X 48.0765, Y 14.6072, Z -3.8333, A 0.000, B 0.000, C 0.000 }
gfCNCPoint3[3573] = {X 47.8320, Y 13.8279, Z -3.8333, A 0.000, B 0.000, C 0.000 }
gfCNCPoint3[3574] = {X 47.7444, Y 13.0158, Z -3.8333, A 0.000, B 0.000, C 0.000 }
gfCNCPoint3[3575] = {X 47.7442, Y 12.1868, Z -3.8333, A 0.000, B 0.000, C 0.000 }
gfCNCPoint3[3576] = {X 47.8485, Y 11.2611, Z -3.8333, A 0.000, B 0.000, C 0.000 }
gfCNCPoint3[3577] = {X 48.1562, Y 10.3819, Z -3.8333, A 0.000, B 0.000, C 0.000 }
gfCNCPoint3[3578] = {X 48.6518, Y 9.5931, Z -3.8333, A 0.000, B 0.000, C 0.000 }
gfCNCPoint3[3579] = {X 49.3105, Y 8.9344, Z -3.8333, A 0.000, B 0.000, C 0.000 }
gfCNCPoint3[3580] = {X 50.0993, Y 8.4388, Z -3.8333, A 0.000, B 0.000, C 0.000 }
gfCNCPoint3[3581] = {X 50.9785, Y 8.1311, Z -3.8333, A 0.000, B 0.000, C 0.000 }
gfCNCPoint3[3582] = {X 51.9042, Y 8.0268, Z -3.8333, A 0.000, B 0.000, C 0.000 }
gfCNCPoint3[3583] = {X 59.6221, Y 8.0268, Z -3.8333, A 0.000, B 0.000, C 0.000 }
gfCNCPoint3[3584] = {X 60.5478, Y 8.1311, Z -3.8333, A 0.000, B 0.000, C 0.000 }
gfCNCPoint3[3585] = {X 61.4271, Y 8.4388, Z -3.8333, A 0.000, B 0.000, C 0.000 }
gfCNCPoint3[3586] = {X 62.2158, Y 8.9344, Z -3.8333, A 0.000, B 0.000, C 0.000 }
gfCNCPoint3[3587] = {X 62.8745, Y 9.5931, Z -3.8333, A 0.000, B 0.000, C 0.000 }
gfCNCPoint3[3588] = {X 63.3702, Y 10.3819, Z -3.8333, A 0.000, B 0.000, C 0.000 }
gfCNCPoint3[3589] = {X 63.6778, Y 11.2611, Z -3.8333, A 0.000, B 0.000, C 0.000 }
gfCNCPoint3[3590] = {X 63.7821, Y 12.1868, Z -3.8333, A 0.000, B 0.000, C 0.000 }
gfCNCPoint3[3591] = {X 63.7821, Y 12.9781, Z -3.8333, A 0.000, B 0.000, C 0.000 }
gfCNCPoint3[3592] = {X 63.6960, Y 13.8202, Z -3.8333, A 0.000, B 0.000, C 0.000 }
gfCNCPoint3[3593] = {X 63.4411, Y 14.6275, Z -3.8333, A 0.000, B 0.000, C 0.000 }
gfCNCPoint3[3594] = {X 63.0282, Y 15.3664, Z -3.8333, A 0.000, B 0.000, C 0.000 }
gfCNCPoint3[3595] = {X 63.2758, Y 16.0199, Z -3.8333, A 0.000, B 0.000, C 0.000 }
gfCNCPoint3[3596] = {X 66.0903, Y 23.4875, Z -3.8333, A 0.000, B 0.000, C 0.000 }
gfCNCPoint3[3597] = {X 72.0600, Y 39.5578, Z -3.8333, A 0.000, B 0.000, C 0.000 }
gfCNCPoint3[3598] = {X 72.3901, Y 40.3881, Z -3.8333, A 0.000, B 0.000, C 0.000 }
gfCNCPoint3[3599] = {X 73.2211, Y 40.8663, Z -3.8333, A 0.000, B 0.000, C 0.000 }
gfCNCPoint3[3600] = {X 73.9205, Y 41.5221, Z -3.8333, A 0.000, B 0.000, C 0.000 }
gfCNCPoint3[3601] = {X 74.4512, Y 42.3206, Z -3.8333, A 0.000, B 0.000, C 0.000 }
gfCNCPoint3[3602] = {X 74.7851, Y 43.2193, Z -3.8333, A 0.000, B 0.000, C 0.000 }
gfCNCPoint3[3603] = {X 74.9043, Y 44.1706, Z -3.8333, A 0.000, B 0.000, C 0.000 }
gfCNCPoint3[3604] = {X 74.9045, Y 45.0000, Z -3.8333, A 0.000, B 0.000, C 0.000 }
gfCNCPoint3[3605] = {X 74.8002, Y 45.9257, Z -3.8333, A 0.000, B 0.000, C 0.000 }
gfCNCPoint3[3606] = {X 74.4925, Y 46.8050, Z -3.8333, A 0.000, B 0.000, C 0.000 }
gfCNCPoint3[3607] = {X 73.9969, Y 47.5937, Z -3.8333, A 0.000, B 0.000, C 0.000 }
gfCNCPoint3[3608] = {X 73.3382, Y 48.2524, Z -3.8333, A 0.000, B 0.000, C 0.000 }
gfCNCPoint3[3609] = {X 72.5494, Y 48.7480, Z -3.8333, A 0.000, B 0.000, C 0.000 }
gfCNCPoint3[3610] = {X 71.6701, Y 49.0557, Z -3.8333, A 0.000, B 0.000, C 0.000 }
gfCNCPoint3[3611] = {X 70.7445, Y 49.1600, Z -3.8333, A 0.000, B 0.000, C 0.000 }
gfCNCPoint3[3612] = {X 64.1851, Y 49.1600, Z -3.8333, A 0.000, B 0.000, C 0.000 }
gfCNCPoint3[3613] = {X 63.2594, Y 49.0557, Z -3.8333, A 0.000, B 0.000, C 0.000 }
gfCNCPoint3[3614] = {X 62.3802, Y 48.7480, Z -3.8333, A 0.000, B 0.000, C 0.000 }
gfCNCPoint3[3615] = {X 61.5914, Y 48.2524, Z -3.8333, A 0.000, B 0.000, C 0.000 }
gfCNCPoint3[3616] = {X 60.9327, Y 47.5937, Z -3.8333, A 0.000, B 0.000, C 0.000 }
gfCNCPoint3[3617] = {X 60.4371, Y 46.8050, Z -3.8333, A 0.000, B 0.000, C 0.000 }
gfCNCPoint3[3618] = {X 60.1294, Y 45.9257, Z -3.8333, A 0.000, B 0.000, C 0.000 }
gfCNCPoint3[3619] = {X 60.0251, Y 45.0000, Z -3.8333, A 0.000, B 0.000, C 0.000 }
gfCNCPoint3[3620] = {X 60.0251, Y 44.2086, Z -3.8333, A 0.000, B 0.000, C 0.000 }
gfCNCPoint3[3621] = {X 60.1142, Y 43.3552, Z -3.8333, A 0.000, B 0.000, C 0.000 }
gfCNCPoint3[3622] = {X 60.3765, Y 42.5383, Z -3.8333, A 0.000, B 0.000, C 0.000 }
gfCNCPoint3[3623] = {X 60.8008, Y 41.7926, Z -3.8333, A 0.000, B 0.000, C 0.000 }
gfCNCPoint3[3624] = {X 60.1189, Y 39.9292, Z -3.8333, A 0.000, B 0.000, C 0.000 }
gfCNCPoint3[3625] = {X 51.9659, Y 39.9292, Z -3.8333, A 0.000, B 0.000, C 0.000 }
gfCNCPoint3[3626] = {X 51.1575, Y 42.1010, Z -3.8333, A 0.000, B 0.000, C 0.000 }
gfCNCPoint3[3627] = {X 51.1992, Y 42.1702, Z -3.8333, A 0.000, B 0.000, C 0.000 }
gfCNCPoint3[3628] = {X 51.4888, Y 42.8047, Z -3.8333, A 0.000, B 0.000, C 0.000 }
gfCNCPoint3[3629] = {X 51.6684, Y 43.4788, Z -3.8333, A 0.000, B 0.000, C 0.000 }
gfCNCPoint3[3630] = {X 51.7328, Y 44.1733, Z -3.8333, A 0.000, B 0.000, C 0.000 }
gfCNCPoint3[3631] = {X 51.7329, Y 45.0000, Z -3.8333, A 0.000, B 0.000, C 0.000 }
gfCNCPoint3[3632] = {X 51.6286, Y 45.9257, Z -3.8333, A 0.000, B 0.000, C 0.000 }
gfCNCPoint3[3633] = {X 51.3210, Y 46.8050, Z -3.8333, A 0.000, B 0.000, C 0.000 }
gfCNCPoint3[3634] = {X 50.8253, Y 47.5937, Z -3.8333, A 0.000, B 0.000, C 0.000 }
gfCNCPoint3[3635] = {X 50.1666, Y 48.2524, Z -3.8333, A 0.000, B 0.000, C 0.000 }
gfCNCPoint3[3636] = {X 49.3779, Y 48.7480, Z -3.8333, A 0.000, B 0.000, C 0.000 }
gfCNCPoint3[3637] = {X 48.4986, Y 49.0557, Z -3.8333, A 0.000, B 0.000, C 0.000 }
gfCNCPoint3[3638] = {X 47.5729, Y 49.1600, Z -3.8333, A 0.000, B 0.000, C 0.000 }
gfCNCPoint3[3639] = {X 40.6393, Y 49.1600, Z -3.8333, A 0.000, B 0.000, C 0.000 }
gfCNCPoint3[3640] = {X 39.7136, Y 49.0557, Z -3.8333, A 0.000, B 0.000, C 0.000 }
gfCNCPoint3[3641] = {X 38.8343, Y 48.7480, Z -3.8333, A 0.000, B 0.000, C 0.000 }
gfCNCPoint3[3642] = {X 38.0456, Y 48.2524, Z -3.8333, A 0.000, B 0.000, C 0.000 }
gfCNCPoint3[3643] = {X 37.3869, Y 47.5937, Z -3.8333, A 0.000, B 0.000, C 0.000 }
gfCNCPoint3[3644] = {X 36.8913, Y 46.8050, Z -3.8333, A 0.000, B 0.000, C 0.000 }
gfCNCPoint3[3645] = {X 36.5836, Y 45.9257, Z -3.8333, A 0.000, B 0.000, C 0.000 }
gfCNCPoint3[3646] = {X 36.4793, Y 45.0000, Z -3.8333, A 0.000, B 0.000, C 0.000 }
gfCNCPoint3[3647] = {X 36.4793, Y 44.2086, Z -3.8333, A 0.000, B 0.000, C 0.000 }
